LIN {X 0,Y 472.91,Z 456.577,A -85,B 0,C 180,E1 22479.324,E2 22479.324} C_VEL
LIN {X 0,Y 472.927,Z 456.575,A -85,B 0,C 180,E1 22475.519,E2 22475.519} C_VEL
LIN {X 0,Y 472.958,Z 456.569,A -85,B 0,C 180,E1 22471.872,E2 22471.872} C_VEL
LIN {X 0,Y 472.951,Z 456.569,A -85,B 0,C 180,E1 22468.195,E2 22468.195} C_VEL
LIN {X 0,Y 472.938,Z 456.573,A -85,B 0,C 180,E1 22464.6,E2 22464.6} C_VEL
LIN {X 0,Y 472.903,Z 456.579,A -85,B 0,C 180,E1 22460.89,E2 22460.89} C_VEL
LIN {X 0,Y 472.947,Z 456.574,A -85,B 0,C 180,E1 22457.263,E2 22457.263} C_VEL
LIN {X 0,Y 472.93,Z 456.574,A -85,B 0,C 180,E1 22453.693,E2 22453.693} C_VEL
LIN {X 0,Y 472.947,Z 456.701,A -85,B 0,C 180,E1 22450.415,E2 22450.415} C_VEL
LIN {X 0,Y 481.637,Z 478.377,A -85,B 0,C 180,E1 22447.531,E2 22447.531} C_VEL
LIN {X 0,Y 487.148,Z 493.23,A -85,B 0,C 180,E1 22445.727,E2 22445.727} C_VEL
LIN {X 0,Y 487.147,Z 498.207,A -85,B 0,C 180,E1 22445.36,E2 22445.36} C_VEL
LIN {X 0,Y 491.021,Z 519.873,A -85,B 0,C 180,E1 22444.656,E2 22444.656} C_VEL
LIN {X 0,Y 490.363,Z 557.478,A -85,B 0,C 180,E1 22444.053,E2 22444.053} C_VEL
LIN {X 0,Y 489.42,Z 565.168,A -85,B 0,C 180,E1 22443.994,E2 22443.994} C_VEL
LIN {X 0,Y 483.858,Z 585.669,A -85,B 0,C 180,E1 22444.081,E2 22444.081} C_VEL
LIN {X 0,Y 483.117,Z 592.27,A -85,B 0,C 180,E1 22444.025,E2 22444.025} C_VEL
LIN {X 0,Y 480.112,Z 758.652,A -85,B 0,C 180,E1 22441.318,E2 22441.318} C_VEL
LIN {X 0,Y 479.264,Z 779.44,A -85,B 0,C 180,E1 22440.773,E2 22440.773} C_VEL
LIN {X 0,Y 478.093,Z 800.27,A -85,B 0,C 180,E1 22439.988,E2 22439.988} C_VEL
LIN {X 0,Y 476.733,Z 819.282,A -85,B 0,C 180,E1 22439.046,E2 22439.046} C_VEL
LIN {X 0,Y 475.203,Z 837.681,A -85,B 0,C 180,E1 22437.907,E2 22437.907} C_VEL
LIN {X 0,Y 473.52,Z 855.537,A -85,B 0,C 180,E1 22436.551,E2 22436.551} C_VEL
LIN {X 0,Y 471.822,Z 872.211,A -85,B 0,C 180,E1 22435.024,E2 22435.024} C_VEL
LIN {X 0,Y 470.132,Z 888.047,A -85,B 0,C 180,E1 22433.301,E2 22433.301} C_VEL
LIN {X 0,Y 468.579,Z 902.793,A -85,B 0,C 180,E1 22431.4,E2 22431.4} C_VEL
LIN {X 0,Y 467.185,Z 916.53,A -85,B 0,C 180,E1 22429.296,E2 22429.296} C_VEL
LIN {X 0,Y 466.056,Z 928.61,A -85,B 0,C 180,E1 22427.092,E2 22427.092} C_VEL
LIN {X 0,Y 465.206,Z 939.007,A -85,B 0,C 180,E1 22424.818,E2 22424.818} C_VEL
LIN {X 0,Y 464.592,Z 947.948,A -85,B 0,C 180,E1 22422.427,E2 22422.427} C_VEL
LIN {X 0,Y 464.221,Z 955.037,A -85,B 0,C 180,E1 22420.047,E2 22420.047} C_VEL
LIN {X 0,Y 464.015,Z 960.75,A -85,B 0,C 180,E1 22417.552,E2 22417.552} C_VEL
LIN {X 0,Y 463.931,Z 964.938,A -85,B 0,C 180,E1 22414.945,E2 22414.945} C_VEL
LIN {X 0,Y 463.912,Z 967.307,A -85,B 0,C 180,E1 22412.47,E2 22412.47} C_VEL
LIN {X 0,Y 463.915,Z 968.138,A -85,B 0,C 180,E1 22409.999,E2 22409.999} C_VEL
LIN {X 0,Y 463.908,Z 967.355,A -85,B 0,C 180,E1 22407.529,E2 22407.529} C_VEL
LIN {X 0,Y 463.932,Z 965.05,A -85,B 0,C 180,E1 22405.054,E2 22405.054} C_VEL
LIN {X 0,Y 464.002,Z 961.169,A -85,B 0,C 180,E1 22402.571,E2 22402.571} C_VEL
LIN {X 0,Y 464.188,Z 955.956,A -85,B 0,C 180,E1 22400.202,E2 22400.202} C_VEL
LIN {X 0,Y 464.549,Z 948.649,A -85,B 0,C 180,E1 22397.696,E2 22397.696} C_VEL
LIN {X 0,Y 465.133,Z 939.852,A -85,B 0,C 180,E1 22395.305,E2 22395.305} C_VEL
LIN {X 0,Y 465.959,Z 929.65,A -85,B 0,C 180,E1 22393.032,E2 22393.032} C_VEL
LIN {X 0,Y 467.101,Z 917.348,A -85,B 0,C 180,E1 22390.752,E2 22390.752} C_VEL
LIN {X 0,Y 468.516,Z 903.403,A -85,B 0,C 180,E1 22388.596,E2 22388.596} C_VEL
LIN {X 0,Y 470.064,Z 888.771,A -85,B 0,C 180,E1 22386.694,E2 22386.694} C_VEL
LIN {X 0,Y 471.702,Z 873.45,A -85,B 0,C 180,E1 22385.007,E2 22385.007} C_VEL
LIN {X 0,Y 473.47,Z 856.09,A -85,B 0,C 180,E1 22383.403,E2 22383.403} C_VEL
LIN {X 0,Y 475.187,Z 837.858,A -85,B 0,C 180,E1 22382.015,E2 22382.015} C_VEL
LIN {X 0,Y 476.704,Z 819.608,A -85,B 0,C 180,E1 22380.881,E2 22380.881} C_VEL
LIN {X 0,Y 478.069,Z 800.671,A -85,B 0,C 180,E1 22379.94,E2 22379.94} C_VEL
LIN {X 0,Y 479.224,Z 780.234,A -85,B 0,C 180,E1 22379.162,E2 22379.162} C_VEL
LIN {X 0,Y 480.082,Z 759.903,A -85,B 0,C 180,E1 22378.618,E2 22378.618} C_VEL
LIN {X 0,Y 481.257,Z 696.258,A -85,B 0,C 180,E1 22377.561,E2 22377.561} C_VEL
LIN {X 0,Y 484.181,Z 528.146,A -85,B 0,C 180,E1 22374.833,E2 22374.833} C_VEL
LIN {X 0,Y 476.532,Z 500.148,A -85,B 0,C 180,E1 22373.647,E2 22373.647} C_VEL
LIN {X 0,Y 476.698,Z 493.601,A -85,B 0,C 180,E1 22372.837,E2 22372.837} C_VEL
LIN {X 0,Y 471.955,Z 477.879,A -85,B 0,C 180,E1 22370.222,E2 22370.222} C_VEL
LIN {X 0,Y 466.792,Z 462.968,A -85,B 0,C 180,E1 22367.566,E2 22367.566} C_VEL
LIN {X 0,Y 465.01,Z 457.558,A -85,B 0,C 180,E1 22366.565,E2 22366.565} C_VEL
LIN {X 0,Y 465.012,Z 457.562,A -85,B 0,C 180,E1 22362.843,E2 22362.843} C_VEL
LIN {X 0,Y 465.017,Z 457.564,A -85,B 0,C 180,E1 22359.209,E2 22359.209} C_VEL
LIN {X 0,Y 465.008,Z 457.58,A -85,B 0,C 180,E1 22355.73,E2 22355.73} C_VEL
LIN {X 0,Y 473.084,Z 479.715,A -85,B 0,C 180,E1 22352.397,E2 22352.397} C_VEL
LIN {X 0,Y 478.097,Z 494.806,A -85,B 0,C 180,E1 22350.262,E2 22350.262} C_VEL
LIN {X 0,Y 476.18,Z 526.834,A -85,B 0,C 180,E1 22346.904,E2 22346.904} C_VEL
LIN {X 0,Y 474.134,Z 562.551,A -85,B 0,C 180,E1 22343.226,E2 22343.226} C_VEL
LIN {X 0,Y 472.412,Z 597.934,A -85,B 0,C 180,E1 22339.635,E2 22339.635} C_VEL
LIN {X 0,Y 471.717,Z 615.117,A -85,B 0,C 180,E1 22337.947,E2 22337.947} C_VEL
LIN {X 0,Y 472.395,Z 621.151,A -85,B 0,C 180,E1 22337.789,E2 22337.789} C_VEL
LIN {X 0,Y 469.651,Z 757.732,A -85,B 0,C 180,E1 22335.181,E2 22335.181} C_VEL
LIN {X 0,Y 469.368,Z 774.573,A -85,B 0,C 180,E1 22334.622,E2 22334.622} C_VEL
LIN {X 0,Y 468.917,Z 789.931,A -85,B 0,C 180,E1 22333.88,E2 22333.88} C_VEL
LIN {X 0,Y 468.342,Z 805.227,A -85,B 0,C 180,E1 22332.891,E2 22332.891} C_VEL
LIN {X 0,Y 467.722,Z 818.619,A -85,B 0,C 180,E1 22331.78,E2 22331.78} C_VEL
LIN {X 0,Y 467.018,Z 832.225,A -85,B 0,C 180,E1 22330.361,E2 22330.361} C_VEL
LIN {X 0,Y 466.406,Z 843.527,A -85,B 0,C 180,E1 22328.879,E2 22328.879} C_VEL
LIN {X 0,Y 465.85,Z 854.094,A -85,B 0,C 180,E1 22327.151,E2 22327.151} C_VEL
LIN {X 0,Y 465.438,Z 862.373,A -85,B 0,C 180,E1 22325.424,E2 22325.424} C_VEL
LIN {X 0,Y 465.125,Z 869.663,A -85,B 0,C 180,E1 22323.451,E2 22323.451} C_VEL
LIN {X 0,Y 464.929,Z 874.839,A -85,B 0,C 180,E1 22321.479,E2 22321.479} C_VEL
LIN {X 0,Y 464.858,Z 878.245,A -85,B 0,C 180,E1 22319.507,E2 22319.507} C_VEL
LIN {X 0,Y 464.842,Z 879.886,A -85,B 0,C 180,E1 22317.535,E2 22317.535} C_VEL
LIN {X 0,Y 464.923,Z 879.826,A -85,B 0,C 180,E1 22315.436,E2 22315.436} C_VEL
LIN {X 0,Y 465.055,Z 877.967,A -85,B 0,C 180,E1 22313.457,E2 22313.457} C_VEL
LIN {X 0,Y 465.317,Z 874.396,A -85,B 0,C 180,E1 22311.474,E2 22311.474} C_VEL
LIN {X 0,Y 465.678,Z 869.023,A -85,B 0,C 180,E1 22309.541,E2 22309.541} C_VEL
LIN {X 0,Y 466.158,Z 862.251,A -85,B 0,C 180,E1 22307.74,E2 22307.74} C_VEL
LIN {X 0,Y 466.757,Z 853.636,A -85,B 0,C 180,E1 22305.992,E2 22305.992} C_VEL
LIN {X 0,Y 467.47,Z 843.493,A -85,B 0,C 180,E1 22304.366,E2 22304.366} C_VEL
LIN {X 0,Y 468.204,Z 832.087,A -85,B 0,C 180,E1 22302.925,E2 22302.925} C_VEL
LIN {X 0,Y 468.927,Z 819.784,A -85,B 0,C 180,E1 22301.669,E2 22301.669} C_VEL
LIN {X 0,Y 469.544,Z 806.42,A -85,B 0,C 180,E1 22300.598,E2 22300.598} C_VEL
LIN {X 0,Y 470.043,Z 792.265,A -85,B 0,C 180,E1 22299.713,E2 22299.713} C_VEL
LIN {X 0,Y 470.359,Z 776.806,A -85,B 0,C 180,E1 22299.011,E2 22299.011} C_VEL
LIN {X 0,Y 470.464,Z 760.839,A -85,B 0,C 180,E1 22298.522,E2 22298.522} C_VEL
LIN {X 0,Y 472.137,Z 707.062,A -85,B 0,C 180,E1 22297.264,E2 22297.264} C_VEL
LIN {X 0,Y 475.823,Z 635.91,A -85,B 0,C 180,E1 22295.48,E2 22295.48} C_VEL
LIN {X 0,Y 479.671,Z 625.998,A -85,B 0,C 180,E1 22294.637,E2 22294.637} C_VEL
LIN {X 0,Y 484.504,Z 596.236,A -85,B 0,C 180,E1 22290.99,E2 22290.99} C_VEL
LIN {X 0,Y 490.347,Z 571.27,A -85,B 0,C 180,E1 22287.708,E2 22287.708} C_VEL
LIN {X 0,Y 496.915,Z 551.415,A -85,B 0,C 180,E1 22284.868,E2 22284.868} C_VEL
LIN {X 0,Y 504.072,Z 536.502,A -85,B 0,C 180,E1 22282.508,E2 22282.508} C_VEL
LIN {X 0,Y 506.427,Z 532.598,A -85,B 0,C 180,E1 22281.76,E2 22281.76} C_VEL
LIN {X 0,Y 506.709,Z 532.003,A -85,B 0,C 180,E1 22281.259,E2 22281.259} C_VEL
LIN {X 0,Y 498.452,Z 544.531,A -85,B 0,C 180,E1 22279.664,E2 22279.664} C_VEL
LIN {X 0,Y 491.821,Z 558.642,A -85,B 0,C 180,E1 22278.022,E2 22278.022} C_VEL
LIN {X 0,Y 487.188,Z 573.707,A -85,B 0,C 180,E1 22276.34,E2 22276.34} C_VEL
LIN {X 0,Y 484.882,Z 588.959,A -85,B 0,C 180,E1 22274.65,E2 22274.65} C_VEL
LIN {X 0,Y 484.928,Z 602.549,A -85,B 0,C 180,E1 22273.122,E2 22273.122} C_VEL
LIN {X 0,Y 487.165,Z 615.999,A -85,B 0,C 180,E1 22271.574,E2 22271.574} C_VEL
LIN {X 0,Y 491.226,Z 627.81,A -85,B 0,C 180,E1 22270.184,E2 22270.184} C_VEL
LIN {X 0,Y 497.098,Z 638.674,A -85,B 0,C 180,E1 22268.871,E2 22268.871} C_VEL
LIN {X 0,Y 504.869,Z 648.854,A -85,B 0,C 180,E1 22267.611,E2 22267.611} C_VEL
LIN {X 0,Y 514.493,Z 658.204,A -85,B 0,C 180,E1 22266.432,E2 22266.432} C_VEL
LIN {X 0,Y 526.445,Z 666.953,A -85,B 0,C 180,E1 22265.302,E2 22265.302} C_VEL
LIN {X 0,Y 516.888,Z 683.64,A -85,B 0,C 180,E1 22264.661,E2 22264.661} C_VEL
LIN {X 0,Y 504.016,Z 702.431,A -85,B 0,C 180,E1 22264.017,E2 22264.017} C_VEL
LIN {X 0,Y 495.13,Z 717.971,A -85,B 0,C 180,E1 22263.387,E2 22263.387} C_VEL
LIN {X 0,Y 488.588,Z 732.528,A -85,B 0,C 180,E1 22262.702,E2 22262.702} C_VEL
LIN {X 0,Y 482.078,Z 749.198,A -85,B 0,C 180,E1 22261.887,E2 22261.887} C_VEL
LIN {X 0,Y 479.563,Z 772.367,A -85,B 0,C 180,E1 22261.674,E2 22261.674} C_VEL
LIN {X 0,Y 478.792,Z 805.933,A -85,B 0,C 180,E1 22261.099,E2 22261.099} C_VEL
LIN {X 0,Y 477.845,Z 826.58,A -85,B 0,C 180,E1 22260.534,E2 22260.534} C_VEL
LIN {X 0,Y 476.592,Z 846.828,A -85,B 0,C 180,E1 22259.747,E2 22259.747} C_VEL
LIN {X 0,Y 475.191,Z 866.116,A -85,B 0,C 180,E1 22258.765,E2 22258.765} C_VEL
LIN {X 0,Y 473.67,Z 884.493,A -85,B 0,C 180,E1 22257.603,E2 22257.603} C_VEL
LIN {X 0,Y 472.077,Z 902.359,A -85,B 0,C 180,E1 22256.233,E2 22256.233} C_VEL
LIN {X 0,Y 470.518,Z 919.286,A -85,B 0,C 180,E1 22254.682,E2 22254.682} C_VEL
LIN {X 0,Y 469.001,Z 935.399,A -85,B 0,C 180,E1 22252.931,E2 22252.931} C_VEL
LIN {X 0,Y 467.587,Z 950.936,A -85,B 0,C 180,E1 22250.923,E2 22250.923} C_VEL
LIN {X 0,Y 466.486,Z 964.207,A -85,B 0,C 180,E1 22248.885,E2 22248.885} C_VEL
LIN {X 0,Y 465.557,Z 976.373,A -85,B 0,C 180,E1 22246.694,E2 22246.694} C_VEL
LIN {X 0,Y 464.832,Z 988.822,A -85,B 0,C 180,E1 22244.068,E2 22244.068} C_VEL
LIN {X 0,Y 464.446,Z 996.901,A -85,B 0,C 180,E1 22242.054,E2 22242.054} C_VEL
LIN {X 0,Y 464.164,Z 1004.554,A -85,B 0,C 180,E1 22239.673,E2 22239.673} C_VEL
LIN {X 0,Y 464.004,Z 1009.721,A -85,B 0,C 180,E1 22237.595,E2 22237.595} C_VEL
LIN {X 0,Y 463.928,Z 1013.749,A -85,B 0,C 180,E1 22235.442,E2 22235.442} C_VEL
LIN {X 0,Y 463.909,Z 1016.649,A -85,B 0,C 180,E1 22232.966,E2 22232.966} C_VEL
LIN {X 0,Y 463.909,Z 1017.726,A -85,B 0,C 180,E1 22230.865,E2 22230.865} C_VEL
LIN {X 0,Y 463.902,Z 1017.607,A -85,B 0,C 180,E1 22228.642,E2 22228.642} C_VEL
LIN {X 0,Y 463.919,Z 1015.695,A -85,B 0,C 180,E1 22226.046,E2 22226.046} C_VEL
LIN {X 0,Y 463.956,Z 1012.73,A -85,B 0,C 180,E1 22223.939,E2 22223.939} C_VEL
LIN {X 0,Y 464.064,Z 1007.975,A -85,B 0,C 180,E1 22221.576,E2 22221.576} C_VEL
LIN {X 0,Y 464.27,Z 1001.352,A -85,B 0,C 180,E1 22219.202,E2 22219.202} C_VEL
LIN {X 0,Y 464.574,Z 994.236,A -85,B 0,C 180,E1 22217.148,E2 22217.148} C_VEL
LIN {X 0,Y 465.136,Z 983.695,A -85,B 0,C 180,E1 22214.669,E2 22214.669} C_VEL
LIN {X 0,Y 465.804,Z 973.255,A -85,B 0,C 180,E1 22212.641,E2 22212.641} C_VEL
LIN {X 0,Y 466.988,Z 957.492,A -85,B 0,C 180,E1 22210.04,E2 22210.04} C_VEL
LIN {X 0,Y 468.228,Z 943.394,A -85,B 0,C 180,E1 22208.057,E2 22208.057} C_VEL
LIN {X 0,Y 469.719,Z 927.266,A -85,B 0,C 180,E1 22206.145,E2 22206.145} C_VEL
LIN {X 0,Y 471.349,Z 909.972,A -85,B 0,C 180,E1 22204.427,E2 22204.427} C_VEL
LIN {X 0,Y 472.911,Z 892.363,A -85,B 0,C 180,E1 22202.964,E2 22202.964} C_VEL
LIN {X 0,Y 474.503,Z 873.954,A -85,B 0,C 180,E1 22201.699,E2 22201.699} C_VEL
LIN {X 0,Y 476.021,Z 854.172,A -85,B 0,C 180,E1 22200.599,E2 22200.599} C_VEL
LIN {X 0,Y 477.32,Z 834.383,A -85,B 0,C 180,E1 22199.741,E2 22199.741} C_VEL
LIN {X 0,Y 478.39,Z 814.17,A -85,B 0,C 180,E1 22199.095,E2 22199.095} C_VEL
LIN {X 0,Y 479.108,Z 792.718,A -85,B 0,C 180,E1 22198.642,E2 22198.642} C_VEL
LIN {X 0,Y 479.824,Z 766.954,A -85,B 0,C 180,E1 22198.252,E2 22198.252} C_VEL
LIN {X 0,Y 480.143,Z 763.831,A -85,B 0,C 180,E1 22198.208,E2 22198.208} C_VEL
LIN {X 0,Y 485.952,Z 747.066,A -85,B 0,C 180,E1 22197.302,E2 22197.302} C_VEL
LIN {X 0,Y 495.745,Z 723.845,A -85,B 0,C 180,E1 22196.197,E2 22196.197} C_VEL
LIN {X 0,Y 504.216,Z 708.095,A -85,B 0,C 180,E1 22195.588,E2 22195.588} C_VEL
LIN {X 0,Y 516.218,Z 689.456,A -85,B 0,C 180,E1 22195.015,E2 22195.015} C_VEL
LIN {X 0,Y 520.11,Z 683.607,A -85,B 0,C 180,E1 22194.848,E2 22194.848} C_VEL
LIN {X 0,Y 528.054,Z 668.908,A -85,B 0,C 180,E1 22194.321,E2 22194.321} C_VEL
LIN {X 0,Y 516.85,Z 661.041,A -85,B 0,C 180,E1 22193.013,E2 22193.013} C_VEL
LIN {X 0,Y 507.468,Z 651.762,A -85,B 0,C 180,E1 22191.644,E2 22191.644} C_VEL
LIN {X 0,Y 500.207,Z 641.723,A -85,B 0,C 180,E1 22190.315,E2 22190.315} C_VEL
LIN {X 0,Y 494.469,Z 630.437,A -85,B 0,C 180,E1 22188.959,E2 22188.959} C_VEL
LIN {X 0,Y 490.186,Z 617.3,A -85,B 0,C 180,E1 22187.534,E2 22187.534} C_VEL
LIN {X 0,Y 487.49,Z 602.313,A -85,B 0,C 180,E1 22186.047,E2 22186.047} C_VEL
LIN {X 0,Y 486.582,Z 585.023,A -85,B 0,C 180,E1 22184.484,E2 22184.484} C_VEL
LIN {X 0,Y 487.699,Z 561.885,A -85,B 0,C 180,E1 22182.574,E2 22182.574} C_VEL
LIN {X 0,Y 490.859,Z 525.783,A -85,B 0,C 180,E1 22179.65,E2 22179.65} C_VEL
LIN {X 0,Y 492.028,Z 513.047,A -85,B 0,C 180,E1 22178.598,E2 22178.598} C_VEL
LIN {X 0,Y 482.947,Z 494.174,A -85,B 0,C 180,E1 22175.72,E2 22175.72} C_VEL
LIN {X 0,Y 473.608,Z 475.089,A -85,B 0,C 180,E1 22172.571,E2 22172.571} C_VEL
LIN {X 0,Y 468.839,Z 465.842,A -85,B 0,C 180,E1 22170.928,E2 22170.928} C_VEL
LIN {X 0,Y 466.513,Z 461.325,A -85,B 0,C 180,E1 22170.101,E2 22170.101} C_VEL
LIN {X 0,Y 465.011,Z 457.678,A -85,B 0,C 180,E1 22169.478,E2 22169.478} C_VEL
LIN {X 0,Y 465.009,Z 457.562,A -85,B 0,C 180,E1 22165.743,E2 22165.743} C_VEL
LIN {X 0,Y 464.994,Z 457.565,A -85,B 0,C 180,E1 22162.104,E2 22162.104} C_VEL
LIN {X 0,Y 464.979,Z 457.567,A -85,B 0,C 180,E1 22158.427,E2 22158.427} C_VEL
LIN {X 0,Y 465.016,Z 457.563,A -85,B 0,C 180,E1 22154.825,E2 22154.825} C_VEL
LIN {X 0,Y 464.988,Z 457.566,A -85,B 0,C 180,E1 22151.158,E2 22151.158} C_VEL
LIN {X 0,Y 465.011,Z 457.561,A -85,B 0,C 180,E1 22147.536,E2 22147.536} C_VEL
LIN {X 0,Y 464.963,Z 457.568,A -85,B 0,C 180,E1 22143.946,E2 22143.946} C_VEL
LIN {X 0,Y 464.993,Z 457.562,A -85,B 0,C 180,E1 22140.246,E2 22140.246} C_VEL
LIN {X 0,Y 465.013,Z 457.564,A -85,B 0,C 180,E1 22136.672,E2 22136.672} C_VEL
LIN {X 0,Y 465.017,Z 457.548,A -85,B 0,C 180,E1 22132.836,E2 22132.836} C_VEL
LIN {X 0,Y 464.994,Z 457.563,A -85,B 0,C 180,E1 22129.218,E2 22129.218} C_VEL
LIN {X 0,Y 464.967,Z 457.562,A -85,B 0,C 180,E1 22125.428,E2 22125.428} C_VEL
LIN {X 0,Y 465.008,Z 457.55,A -85,B 0,C 180,E1 22121.833,E2 22121.833} C_VEL
LIN {X 0,Y 465.003,Z 457.555,A -85,B 0,C 180,E1 22118.162,E2 22118.162} C_VEL
LIN {X 0,Y 465.013,Z 457.561,A -85,B 0,C 180,E1 22114.53,E2 22114.53} C_VEL
LIN {X 0,Y 464.97,Z 457.568,A -85,B 0,C 180,E1 22110.923,E2 22110.923} C_VEL
LIN {X 0,Y 464.988,Z 457.566,A -85,B 0,C 180,E1 22107.189,E2 22107.189} C_VEL
LIN {X 0,Y 465.016,Z 457.565,A -85,B 0,C 180,E1 22103.528,E2 22103.528} C_VEL
LIN {X 0,Y 465.022,Z 457.556,A -85,B 0,C 180,E1 22099.755,E2 22099.755} C_VEL
LIN {X 0,Y 464.998,Z 457.561,A -85,B 0,C 180,E1 22096.081,E2 22096.081} C_VEL
LIN {X 0,Y 464.967,Z 457.569,A -85,B 0,C 180,E1 22092.291,E2 22092.291} C_VEL
LIN {X 0,Y 465.006,Z 457.62,A -85,B 0,C 180,E1 22091.144,E2 22091.144} C_VEL
LIN {X 0,Y 466.275,Z 461.028,A -85,B 0,C 180,E1 22090.683,E2 22090.683} C_VEL
LIN {X 0,Y 473.647,Z 478.764,A -85,B 0,C 180,E1 22088.253,E2 22088.253} C_VEL
LIN {X 0,Y 480.276,Z 496.419,A -85,B 0,C 180,E1 22086.077,E2 22086.077} C_VEL
LIN {X 0,Y 480.45,Z 498.811,A -85,B 0,C 180,E1 22085.923,E2 22085.923} C_VEL
LIN {X 0,Y 484.443,Z 521.253,A -85,B 0,C 180,E1 22085.177,E2 22085.177} C_VEL
LIN {X 0,Y 483.117,Z 592.27,A -85,B 0,C 180,E1 22084.025,E2 22084.025} C_VEL
LIN {X 0,Y 482.157,Z 599.961,A -85,B 0,C 180,E1 22083.966,E2 22083.966} C_VEL
LIN {X 0,Y 476.58,Z 620.456,A -85,B 0,C 180,E1 22084.055,E2 22084.055} C_VEL
LIN {X 0,Y 475.826,Z 627.058,A -85,B 0,C 180,E1 22083.999,E2 22083.999} C_VEL
LIN {X 0,Y 473.287,Z 759.334,A -85,B 0,C 180,E1 22081.813,E2 22081.813} C_VEL
LIN {X 0,Y 472.398,Z 779.954,A -85,B 0,C 180,E1 22081.264,E2 22081.264} C_VEL
LIN {X 0,Y 471.167,Z 800.633,A -85,B 0,C 180,E1 22080.475,E2 22080.475} C_VEL
LIN {X 0,Y 469.702,Z 819.966,A -85,B 0,C 180,E1 22079.504,E2 22079.504} C_VEL
LIN {X 0,Y 468.075,Z 838.339,A -85,B 0,C 180,E1 22078.348,E2 22078.348} C_VEL
LIN {X 0,Y 466.286,Z 856.248,A -85,B 0,C 180,E1 22076.968,E2 22076.968} C_VEL
LIN {X 0,Y 464.421,Z 873.405,A -85,B 0,C 180,E1 22075.367,E2 22075.367} C_VEL
LIN {X 0,Y 462.695,Z 888.451,A -85,B 0,C 180,E1 22073.699,E2 22073.699} C_VEL
LIN {X 0,Y 461.032,Z 903.202,A -85,B 0,C 180,E1 22071.768,E2 22071.768} C_VEL
LIN {X 0,Y 459.575,Z 916.502,A -85,B 0,C 180,E1 22069.707,E2 22069.707} C_VEL
LIN {X 0,Y 458.366,Z 928.408,A -85,B 0,C 180,E1 22067.519,E2 22067.519} C_VEL
LIN {X 0,Y 457.418,Z 938.91,A -85,B 0,C 180,E1 22065.206,E2 22065.206} C_VEL
LIN {X 0,Y 456.728,Z 947.92,A -85,B 0,C 180,E1 22062.773,E2 22062.773} C_VEL
LIN {X 0,Y 456.29,Z 955.25,A -85,B 0,C 180,E1 22060.299,E2 22060.299} C_VEL
LIN {X 0,Y 456.064,Z 960.918,A -85,B 0,C 180,E1 22057.812,E2 22057.812} C_VEL
LIN {X 0,Y 455.949,Z 965.044,A -85,B 0,C 180,E1 22055.284,E2 22055.284} C_VEL
LIN {X 0,Y 455.926,Z 967.588,A -85,B 0,C 180,E1 22052.765,E2 22052.765} C_VEL
LIN {X 0,Y 455.925,Z 968.528,A -85,B 0,C 180,E1 22050.125,E2 22050.125} C_VEL
LIN {X 0,Y 455.92,Z 967.832,A -85,B 0,C 180,E1 22047.611,E2 22047.611} C_VEL
LIN {X 0,Y 455.948,Z 965.462,A -85,B 0,C 180,E1 22044.967,E2 22044.967} C_VEL
LIN {X 0,Y 456.035,Z 961.58,A -85,B 0,C 180,E1 22042.44,E2 22042.44} C_VEL
LIN {X 0,Y 456.247,Z 956.368,A -85,B 0,C 180,E1 22040.03,E2 22040.03} C_VEL
LIN {X 0,Y 456.649,Z 949.061,A -85,B 0,C 180,E1 22037.48,E2 22037.48} C_VEL
LIN {X 0,Y 457.295,Z 940.262,A -85,B 0,C 180,E1 22035.048,E2 22035.048} C_VEL
LIN {X 0,Y 458.195,Z 930.057,A -85,B 0,C 180,E1 22032.735,E2 22032.735} C_VEL
LIN {X 0,Y 459.435,Z 917.751,A -85,B 0,C 180,E1 22030.418,E2 22030.418} C_VEL
LIN {X 0,Y 460.965,Z 903.801,A -85,B 0,C 180,E1 22028.228,E2 22028.228} C_VEL
LIN {X 0,Y 462.668,Z 888.727,A -85,B 0,C 180,E1 22026.244,E2 22026.244} C_VEL
LIN {X 0,Y 464.468,Z 872.95,A -85,B 0,C 180,E1 22024.497,E2 22024.497} C_VEL
LIN {X 0,Y 466.265,Z 856.46,A -85,B 0,C 180,E1 22022.959,E2 22022.959} C_VEL
LIN {X 0,Y 468.09,Z 838.221,A -85,B 0,C 180,E1 22021.553,E2 22021.553} C_VEL
LIN {X 0,Y 469.703,Z 819.96,A -85,B 0,C 180,E1 22020.405,E2 22020.405} C_VEL
LIN {X 0,Y 471.159,Z 800.795,A -85,B 0,C 180,E1 22019.442,E2 22019.442} C_VEL
LIN {X 0,Y 472.394,Z 780.039,A -85,B 0,C 180,E1 22018.648,E2 22018.648} C_VEL
LIN {X 0,Y 473.289,Z 759.337,A -85,B 0,C 180,E1 22018.097,E2 22018.097} C_VEL
LIN {X 0,Y 476.178,Z 607.269,A -85,B 0,C 180,E1 22015.583,E2 22015.583} C_VEL
LIN {X 0,Y 477.536,Z 529.583,A -85,B 0,C 180,E1 22014.292,E2 22014.292} C_VEL
LIN {X 0,Y 469.619,Z 500.423,A -85,B 0,C 180,E1 22013.017,E2 22013.017} C_VEL
LIN {X 0,Y 469.622,Z 496.818,A -85,B 0,C 180,E1 22012.575,E2 22012.575} C_VEL
LIN {X 0,Y 464.912,Z 481.204,A -85,B 0,C 180,E1 22009.963,E2 22009.963} C_VEL
LIN {X 0,Y 459.304,Z 464.811,A -85,B 0,C 180,E1 22007.007,E2 22007.007} C_VEL
LIN {X 0,Y 457.05,Z 458.55,A -85,B 0,C 180,E1 22005.797,E2 22005.797} C_VEL
LIN {X 0,Y 457.06,Z 458.547,A -85,B 0,C 180,E1 22002.021,E2 22002.021} C_VEL
LIN {X 0,Y 457.074,Z 458.552,A -85,B 0,C 180,E1 21998.408,E2 21998.408} C_VEL
LIN {X 0,Y 457.096,Z 458.744,A -85,B 0,C 180,E1 21996.392,E2 21996.392} C_VEL
LIN {X 0,Y 465.159,Z 480.489,A -85,B 0,C 180,E1 21993.037,E2 21993.037} C_VEL
LIN {X 0,Y 470.961,Z 497.618,A -85,B 0,C 180,E1 21990.562,E2 21990.562} C_VEL
LIN {X 0,Y 468.998,Z 528.902,A -85,B 0,C 180,E1 21987.25,E2 21987.25} C_VEL
LIN {X 0,Y 466.848,Z 564.434,A -85,B 0,C 180,E1 21983.556,E2 21983.556} C_VEL
LIN {X 0,Y 465.013,Z 599.849,A -85,B 0,C 180,E1 21979.926,E2 21979.926} C_VEL
LIN {X 0,Y 464.303,Z 616.005,A -85,B 0,C 180,E1 21978.32,E2 21978.32} C_VEL
LIN {X 0,Y 465.008,Z 622.209,A -85,B 0,C 180,E1 21978.154,E2 21978.154} C_VEL
LIN {X 0,Y 462.034,Z 758.851,A -85,B 0,C 180,E1 21975.461,E2 21975.461} C_VEL
LIN {X 0,Y 461.725,Z 775.984,A -85,B 0,C 180,E1 21974.877,E2 21974.877} C_VEL
LIN {X 0,Y 461.246,Z 791.353,A -85,B 0,C 180,E1 21974.115,E2 21974.115} C_VEL
LIN {X 0,Y 460.641,Z 806.561,A -85,B 0,C 180,E1 21973.11,E2 21973.11} C_VEL
LIN {X 0,Y 459.952,Z 820.55,A -85,B 0,C 180,E1 21971.918,E2 21971.918} C_VEL
LIN {X 0,Y 459.245,Z 833.485,A -85,B 0,C 180,E1 21970.538,E2 21970.538} C_VEL
LIN {X 0,Y 458.587,Z 844.985,A -85,B 0,C 180,E1 21969,E2 21969} C_VEL
LIN {X 0,Y 458.01,Z 855.345,A -85,B 0,C 180,E1 21967.274,E2 21967.274} C_VEL
LIN {X 0,Y 457.572,Z 863.623,A -85,B 0,C 180,E1 21965.517,E2 21965.517} C_VEL
LIN {X 0,Y 457.239,Z 870.93,A -85,B 0,C 180,E1 21963.511,E2 21963.511} C_VEL
LIN {X 0,Y 457.032,Z 876.115,A -85,B 0,C 180,E1 21961.505,E2 21961.505} C_VEL
LIN {X 0,Y 456.958,Z 879.536,A -85,B 0,C 180,E1 21959.499,E2 21959.499} C_VEL
LIN {X 0,Y 456.946,Z 881.179,A -85,B 0,C 180,E1 21957.492,E2 21957.492} C_VEL
LIN {X 0,Y 457.038,Z 881.126,A -85,B 0,C 180,E1 21955.357,E2 21955.357} C_VEL
LIN {X 0,Y 457.194,Z 879.271,A -85,B 0,C 180,E1 21953.344,E2 21953.344} C_VEL
LIN {X 0,Y 457.49,Z 875.714,A -85,B 0,C 180,E1 21951.327,E2 21951.327} C_VEL
LIN {X 0,Y 457.879,Z 870.565,A -85,B 0,C 180,E1 21949.431,E2 21949.431} C_VEL
LIN {X 0,Y 458.429,Z 863.572,A -85,B 0,C 180,E1 21947.53,E2 21947.53} C_VEL
LIN {X 0,Y 459.088,Z 854.863,A -85,B 0,C 180,E1 21945.74,E2 21945.74} C_VEL
LIN {X 0,Y 459.864,Z 844.801,A -85,B 0,C 180,E1 21944.1,E2 21944.1} C_VEL
LIN {X 0,Y 460.709,Z 832.889,A -85,B 0,C 180,E1 21942.573,E2 21942.573} C_VEL
LIN {X 0,Y 461.444,Z 821.109,A -85,B 0,C 180,E1 21941.361,E2 21941.361} C_VEL
LIN {X 0,Y 462.144,Z 806.943,A -85,B 0,C 180,E1 21940.216,E2 21940.216} C_VEL
LIN {X 0,Y 462.661,Z 793.229,A -85,B 0,C 180,E1 21939.353,E2 21939.353} C_VEL
LIN {X 0,Y 463.025,Z 776.838,A -85,B 0,C 180,E1 21938.605,E2 21938.605} C_VEL
LIN {X 0,Y 463.119,Z 759.97,A -85,B 0,C 180,E1 21938.105,E2 21938.105} C_VEL
LIN {X 0,Y 465.355,Z 702.161,A -85,B 0,C 180,E1 21936.667,E2 21936.667} C_VEL
LIN {X 0,Y 469.061,Z 638.911,A -85,B 0,C 180,E1 21935.002,E2 21935.002} C_VEL
LIN {X 0,Y 473.322,Z 628.666,A -85,B 0,C 180,E1 21934.146,E2 21934.146} C_VEL
LIN {X 0,Y 478.491,Z 599.761,A -85,B 0,C 180,E1 21930.521,E2 21930.521} C_VEL
LIN {X 0,Y 484.675,Z 575.767,A -85,B 0,C 180,E1 21927.283,E2 21927.283} C_VEL
LIN {X 0,Y 491.407,Z 557.225,A -85,B 0,C 180,E1 21924.558,E2 21924.558} C_VEL
LIN {X 0,Y 498.613,Z 543.248,A -85,B 0,C 180,E1 21922.294,E2 21922.294} C_VEL
LIN {X 0,Y 501.214,Z 539.311,A -85,B 0,C 180,E1 21921.536,E2 21921.536} C_VEL
LIN {X 0,Y 492.979,Z 551.27,A -85,B 0,C 180,E1 21919.989,E2 21919.989} C_VEL
LIN {X 0,Y 485.998,Z 565.215,A -85,B 0,C 180,E1 21918.316,E2 21918.316} C_VEL
LIN {X 0,Y 481.3,Z 579.554,A -85,B 0,C 180,E1 21916.644,E2 21916.644} C_VEL
LIN {X 0,Y 478.822,Z 594.617,A -85,B 0,C 180,E1 21914.895,E2 21914.895} C_VEL
LIN {X 0,Y 478.803,Z 608.074,A -85,B 0,C 180,E1 21913.302,E2 21913.302} C_VEL
LIN {X 0,Y 481.079,Z 621.491,A -85,B 0,C 180,E1 21911.689,E2 21911.689} C_VEL
LIN {X 0,Y 485.242,Z 633.346,A -85,B 0,C 180,E1 21910.233,E2 21910.233} C_VEL
LIN {X 0,Y 491.493,Z 644.617,A -85,B 0,C 180,E1 21908.818,E2 21908.818} C_VEL
LIN {X 0,Y 499.335,Z 654.66,A -85,B 0,C 180,E1 21907.539,E2 21907.539} C_VEL
LIN {X 0,Y 509.66,Z 664.499,A -85,B 0,C 180,E1 21906.264,E2 21906.264} C_VEL
LIN {X 0,Y 516.744,Z 669.987,A -85,B 0,C 180,E1 21905.548,E2 21905.548} C_VEL
LIN {X 0,Y 510.804,Z 680.638,A -85,B 0,C 180,E1 21905.134,E2 21905.134} C_VEL
LIN {X 0,Y 497.845,Z 699.542,A -85,B 0,C 180,E1 21904.498,E2 21904.498} C_VEL
LIN {X 0,Y 488.408,Z 716.01,A -85,B 0,C 180,E1 21903.838,E2 21903.838} C_VEL
LIN {X 0,Y 481.438,Z 731.474,A -85,B 0,C 180,E1 21903.108,E2 21903.108} C_VEL
LIN {X 0,Y 475.786,Z 745.763,A -85,B 0,C 180,E1 21902.416,E2 21902.416} C_VEL
LIN {X 0,Y 472.889,Z 770.51,A -85,B 0,C 180,E1 21902.204,E2 21902.204} C_VEL
LIN {X 0,Y 471.954,Z 805.073,A -85,B 0,C 180,E1 21901.617,E2 21901.617} C_VEL
LIN {X 0,Y 470.941,Z 826.01,A -85,B 0,C 180,E1 21901.04,E2 21901.04} C_VEL
LIN {X 0,Y 469.578,Z 846.478,A -85,B 0,C 180,E1 21900.237,E2 21900.237} C_VEL
LIN {X 0,Y 468.079,Z 865.821,A -85,B 0,C 180,E1 21899.24,E2 21899.24} C_VEL
LIN {X 0,Y 466.369,Z 885.021,A -85,B 0,C 180,E1 21898.004,E2 21898.004} C_VEL
LIN {X 0,Y 464.638,Z 903.003,A -85,B 0,C 180,E1 21896.59,E2 21896.59} C_VEL
LIN {X 0,Y 462.93,Z 920.12,A -85,B 0,C 180,E1 21894.977,E2 21894.977} C_VEL
LIN {X 0,Y 461.334,Z 935.815,A -85,B 0,C 180,E1 21893.228,E2 21893.228} C_VEL
LIN {X 0,Y 459.812,Z 951.436,A -85,B 0,C 180,E1 21891.16,E2 21891.16} C_VEL
LIN {X 0,Y 458.576,Z 965.387,A -85,B 0,C 180,E1 21888.959,E2 21888.959} C_VEL
LIN {X 0,Y 457.563,Z 977.708,A -85,B 0,C 180,E1 21886.635,E2 21886.635} C_VEL
LIN {X 0,Y 456.926,Z 987.365,A -85,B 0,C 180,E1 21884.446,E2 21884.446} C_VEL
LIN {X 0,Y 456.434,Z 997.439,A -85,B 0,C 180,E1 21881.709,E2 21881.709} C_VEL
LIN {X 0,Y 456.185,Z 1004.243,A -85,B 0,C 180,E1 21879.462,E2 21879.462} C_VEL
LIN {X 0,Y 456.05,Z 1009.104,A -85,B 0,C 180,E1 21877.433,E2 21877.433} C_VEL
LIN {X 0,Y 455.997,Z 1013.486,A -85,B 0,C 180,E1 21874.906,E2 21874.906} C_VEL
LIN {X 0,Y 455.983,Z 1015.796,A -85,B 0,C 180,E1 21872.64,E2 21872.64} C_VEL
LIN {X 0,Y 455.972,Z 1016.749,A -85,B 0,C 180,E1 21870.503,E2 21870.503} C_VEL
LIN {X 0,Y 455.978,Z 1016.201,A -85,B 0,C 180,E1 21867.864,E2 21867.864} C_VEL
LIN {X 0,Y 455.982,Z 1014.327,A -85,B 0,C 180,E1 21865.725,E2 21865.725} C_VEL
LIN {X 0,Y 456.016,Z 1011.232,A -85,B 0,C 180,E1 21863.58,E2 21863.58} C_VEL
LIN {X 0,Y 456.121,Z 1005.905,A -85,B 0,C 180,E1 21861.047,E2 21861.047} C_VEL
LIN {X 0,Y 456.321,Z 999.801,A -85,B 0,C 180,E1 21858.883,E2 21858.883} C_VEL
LIN {X 0,Y 456.66,Z 992.274,A -85,B 0,C 180,E1 21856.71,E2 21856.71} C_VEL
LIN {X 0,Y 457.336,Z 980.719,A -85,B 0,C 180,E1 21854.011,E2 21854.011} C_VEL
LIN {X 0,Y 458.222,Z 968.816,A -85,B 0,C 180,E1 21851.656,E2 21851.656} C_VEL
LIN {X 0,Y 459.357,Z 955.74,A -85,B 0,C 180,E1 21849.486,E2 21849.486} C_VEL
LIN {X 0,Y 460.743,Z 941.445,A -85,B 0,C 180,E1 21847.48,E2 21847.48} C_VEL
LIN {X 0,Y 462.31,Z 925.666,A -85,B 0,C 180,E1 21845.602,E2 21845.602} C_VEL
LIN {X 0,Y 464.102,Z 908.208,A -85,B 0,C 180,E1 21843.86,E2 21843.86} C_VEL
LIN {X 0,Y 465.82,Z 890.344,A -85,B 0,C 180,E1 21842.379,E2 21842.379} C_VEL
LIN {X 0,Y 467.521,Z 871.56,A -85,B 0,C 180,E1 21841.097,E2 21841.097} C_VEL
LIN {X 0,Y 469.033,Z 853.102,A -85,B 0,C 180,E1 21840.078,E2 21840.078} C_VEL
LIN {X 0,Y 470.425,Z 832.848,A -85,B 0,C 180,E1 21839.202,E2 21839.202} C_VEL
LIN {X 0,Y 471.566,Z 812.575,A -85,B 0,C 180,E1 21838.562,E2 21838.562} C_VEL
LIN {X 0,Y 472.293,Z 791.352,A -85,B 0,C 180,E1 21838.117,E2 21838.117} C_VEL
LIN {X 0,Y 473.023,Z 766.977,A -85,B 0,C 180,E1 21837.745,E2 21837.745} C_VEL
LIN {X 0,Y 473.561,Z 761.818,A -85,B 0,C 180,E1 21837.677,E2 21837.677} C_VEL
LIN {X 0,Y 479.309,Z 745.604,A -85,B 0,C 180,E1 21836.799,E2 21836.799} C_VEL
LIN {X 0,Y 488.945,Z 723.093,A -85,B 0,C 180,E1 21835.705,E2 21835.705} C_VEL
LIN {X 0,Y 497.672,Z 706.799,A -85,B 0,C 180,E1 21835.07,E2 21835.07} C_VEL
LIN {X 0,Y 509.741,Z 687.982,A -85,B 0,C 180,E1 21834.491,E2 21834.491} C_VEL
LIN {X 0,Y 514.103,Z 681.452,A -85,B 0,C 180,E1 21834.307,E2 21834.307} C_VEL
LIN {X 0,Y 518.82,Z 672.394,A -85,B 0,C 180,E1 21833.968,E2 21833.968} C_VEL
LIN {X 0,Y 508.894,Z 664.689,A -85,B 0,C 180,E1 21832.724,E2 21832.724} C_VEL
LIN {X 0,Y 499.684,Z 654.89,A -85,B 0,C 180,E1 21831.295,E2 21831.295} C_VEL
LIN {X 0,Y 492.122,Z 643.464,A -85,B 0,C 180,E1 21829.812,E2 21829.812} C_VEL
LIN {X 0,Y 486.671,Z 631.501,A -85,B 0,C 180,E1 21828.403,E2 21828.403} C_VEL
LIN {X 0,Y 482.622,Z 617.214,A -85,B 0,C 180,E1 21826.87,E2 21826.87} C_VEL
LIN {X 0,Y 480.342,Z 601.127,A -85,B 0,C 180,E1 21825.287,E2 21825.287} C_VEL
LIN {X 0,Y 479.951,Z 582.116,A -85,B 0,C 180,E1 21823.595,E2 21823.595} C_VEL
LIN {X 0,Y 484.516,Z 527.597,A -85,B 0,C 180,E1 21819.112,E2 21819.112} C_VEL
LIN {X 0,Y 485.464,Z 516.754,A -85,B 0,C 180,E1 21818.202,E2 21818.202} C_VEL
LIN {X 0,Y 475.659,Z 496.26,A -85,B 0,C 180,E1 21815.02,E2 21815.02} C_VEL
LIN {X 0,Y 467.32,Z 479.48,A -85,B 0,C 180,E1 21812.191,E2 21812.191} C_VEL
LIN {X 0,Y 460.973,Z 466.923,A -85,B 0,C 180,E1 21809.925,E2 21809.925} C_VEL
LIN {X 0,Y 459.079,Z 462.973,A -85,B 0,C 180,E1 21809.2,E2 21809.2} C_VEL
LIN {X 0,Y 457.351,Z 460.015,A -85,B 0,C 180,E1 21808.605,E2 21808.605} C_VEL
LIN {X 0,Y 457.041,Z 458.555,A -85,B 0,C 180,E1 21808.341,E2 21808.341} C_VEL
LIN {X 0,Y 457.072,Z 458.551,A -85,B 0,C 180,E1 21804.697,E2 21804.697} C_VEL
LIN {X 0,Y 457.045,Z 458.556,A -85,B 0,C 180,E1 21801.025,E2 21801.025} C_VEL
LIN {X 0,Y 457.062,Z 458.553,A -85,B 0,C 180,E1 21797.308,E2 21797.308} C_VEL
LIN {X 0,Y 457.065,Z 458.554,A -85,B 0,C 180,E1 21793.666,E2 21793.666} C_VEL
LIN {X 0,Y 457.061,Z 458.556,A -85,B 0,C 180,E1 21789.824,E2 21789.824} C_VEL
LIN {X 0,Y 457.06,Z 458.555,A -85,B 0,C 180,E1 21786.153,E2 21786.153} C_VEL
LIN {X 0,Y 457.025,Z 458.556,A -85,B 0,C 180,E1 21782.382,E2 21782.382} C_VEL
LIN {X 0,Y 457.074,Z 458.549,A -85,B 0,C 180,E1 21778.746,E2 21778.746} C_VEL
LIN {X 0,Y 457.044,Z 458.554,A -85,B 0,C 180,E1 21775.105,E2 21775.105} C_VEL
LIN {X 0,Y 457.071,Z 458.538,A -85,B 0,C 180,E1 21771.445,E2 21771.445} C_VEL
LIN {X 0,Y 457.037,Z 458.544,A -85,B 0,C 180,E1 21767.748,E2 21767.748} C_VEL
LIN {X 0,Y 457.052,Z 458.552,A -85,B 0,C 180,E1 21764,E2 21764} C_VEL
LIN {X 0,Y 457.076,Z 458.547,A -85,B 0,C 180,E1 21760.313,E2 21760.313} C_VEL
LIN {X 0,Y 457.07,Z 458.542,A -85,B 0,C 180,E1 21756.538,E2 21756.538} C_VEL
LIN {X 0,Y 457.06,Z 458.543,A -85,B 0,C 180,E1 21752.915,E2 21752.915} C_VEL
LIN {X 0,Y 457.026,Z 458.547,A -85,B 0,C 180,E1 21749.207,E2 21749.207} C_VEL
LIN {X 0,Y 457.069,Z 458.545,A -85,B 0,C 180,E1 21745.557,E2 21745.557} C_VEL
LIN {X 0,Y 457.054,Z 458.546,A -85,B 0,C 180,E1 21741.909,E2 21741.909} C_VEL
LIN {X 0,Y 457.077,Z 458.548,A -85,B 0,C 180,E1 21738.239,E2 21738.239} C_VEL
LIN {X 0,Y 457.039,Z 458.554,A -85,B 0,C 180,E1 21734.505,E2 21734.505} C_VEL
LIN {X 0,Y 457.075,Z 458.737,A -85,B 0,C 180,E1 21731.889,E2 21731.889} C_VEL
LIN {X 0,Y 458.625,Z 462.373,A -85,B 0,C 180,E1 21731.366,E2 21731.366} C_VEL
LIN {X 0,Y 467.098,Z 482.792,A -85,B 0,C 180,E1 21728.528,E2 21728.528} C_VEL
LIN {X 0,Y 473.129,Z 498.641,A -85,B 0,C 180,E1 21726.577,E2 21726.577} C_VEL
LIN {X 0,Y 474.178,Z 501.412,A -85,B 0,C 180,E1 21726.431,E2 21726.431} C_VEL
LIN {X 0,Y 477.906,Z 522.604,A -85,B 0,C 180,E1 21725.711,E2 21725.711} C_VEL
LIN {X 0,Y 475.826,Z 627.058,A -85,B 0,C 180,E1 21723.999,E2 21723.999} C_VEL
LIN {X 0,Y 474.851,Z 634.747,A -85,B 0,C 180,E1 21723.941,E2 21723.941} C_VEL
LIN {X 0,Y 469.266,Z 655.235,A -85,B 0,C 180,E1 21724.032,E2 21724.032} C_VEL
LIN {X 0,Y 468.504,Z 661.834,A -85,B 0,C 180,E1 21723.975,E2 21723.975} C_VEL
LIN {X 0,Y 466.499,Z 760.03,A -85,B 0,C 180,E1 21722.322,E2 21722.322} C_VEL
LIN {X 0,Y 465.559,Z 780.627,A -85,B 0,C 180,E1 21721.765,E2 21721.765} C_VEL
LIN {X 0,Y 464.276,Z 801.002,A -85,B 0,C 180,E1 21720.977,E2 21720.977} C_VEL
LIN {X 0,Y 462.725,Z 820.429,A -85,B 0,C 180,E1 21719.989,E2 21719.989} C_VEL
LIN {X 0,Y 460.976,Z 839.001,A -85,B 0,C 180,E1 21718.803,E2 21718.803} C_VEL
LIN {X 0,Y 459.079,Z 856.956,A -85,B 0,C 180,E1 21717.398,E2 21717.398} C_VEL
LIN {X 0,Y 457.052,Z 874.453,A -85,B 0,C 180,E1 21715.736,E2 21715.736} C_VEL
LIN {X 0,Y 455.134,Z 890.152,A -85,B 0,C 180,E1 21713.951,E2 21713.951} C_VEL
LIN {X 0,Y 453.395,Z 904.51,A -85,B 0,C 180,E1 21712.017,E2 21712.017} C_VEL
LIN {X 0,Y 451.801,Z 918.049,A -85,B 0,C 180,E1 21709.856,E2 21709.856} C_VEL
LIN {X 0,Y 450.49,Z 930.054,A -85,B 0,C 180,E1 21707.568,E2 21707.568} C_VEL
LIN {X 0,Y 449.496,Z 940.336,A -85,B 0,C 180,E1 21705.217,E2 21705.217} C_VEL
LIN {X 0,Y 448.778,Z 949.207,A -85,B 0,C 180,E1 21702.742,E2 21702.742} C_VEL
LIN {X 0,Y 448.313,Z 956.551,A -85,B 0,C 180,E1 21700.147,E2 21700.147} C_VEL
LIN {X 0,Y 448.077,Z 961.824,A -85,B 0,C 180,E1 21697.694,E2 21697.694} C_VEL
LIN {X 0,Y 447.963,Z 965.765,A -85,B 0,C 180,E1 21695.122,E2 21695.122} C_VEL
LIN {X 0,Y 447.936,Z 968.131,A -85,B 0,C 180,E1 21692.558,E2 21692.558} C_VEL
LIN {X 0,Y 447.937,Z 968.961,A -85,B 0,C 180,E1 21689.999,E2 21689.999} C_VEL
LIN {X 0,Y 447.932,Z 968.178,A -85,B 0,C 180,E1 21687.441,E2 21687.441} C_VEL
LIN {X 0,Y 447.964,Z 965.873,A -85,B 0,C 180,E1 21684.877,E2 21684.877} C_VEL
LIN {X 0,Y 448.079,Z 961.801,A -85,B 0,C 180,E1 21682.205,E2 21682.205} C_VEL
LIN {X 0,Y 448.319,Z 956.439,A -85,B 0,C 180,E1 21679.722,E2 21679.722} C_VEL
LIN {X 0,Y 448.789,Z 949.072,A -85,B 0,C 180,E1 21677.126,E2 21677.126} C_VEL
LIN {X 0,Y 449.564,Z 939.674,A -85,B 0,C 180,E1 21674.52,E2 21674.52} C_VEL
LIN {X 0,Y 450.582,Z 929.231,A -85,B 0,C 180,E1 21672.167,E2 21672.167} C_VEL
LIN {X 0,Y 451.877,Z 917.404,A -85,B 0,C 180,E1 21669.942,E2 21669.942} C_VEL
LIN {X 0,Y 453.443,Z 904.133,A -85,B 0,C 180,E1 21667.838,E2 21667.838} C_VEL
LIN {X 0,Y 455.269,Z 889.01,A -85,B 0,C 180,E1 21665.82,E2 21665.82} C_VEL
LIN {X 0,Y 457.174,Z 873.334,A -85,B 0,C 180,E1 21664.061,E2 21664.061} C_VEL
LIN {X 0,Y 459.092,Z 856.84,A -85,B 0,C 180,E1 21662.501,E2 21662.501} C_VEL
LIN {X 0,Y 461.025,Z 838.594,A -85,B 0,C 180,E1 21661.076,E2 21661.076} C_VEL
LIN {X 0,Y 462.737,Z 820.322,A -85,B 0,C 180,E1 21659.914,E2 21659.914} C_VEL
LIN {X 0,Y 464.265,Z 801.229,A -85,B 0,C 180,E1 21658.943,E2 21658.943} C_VEL
LIN {X 0,Y 465.579,Z 780.352,A -85,B 0,C 180,E1 21658.136,E2 21658.136} C_VEL
LIN {X 0,Y 466.516,Z 759.581,A -85,B 0,C 180,E1 21657.578,E2 21657.578} C_VEL
LIN {X 0,Y 471.179,Z 531.965,A -85,B 0,C 180,E1 21653.774,E2 21653.774} C_VEL
LIN {X 0,Y 462.755,Z 500.804,A -85,B 0,C 180,E1 21652.381,E2 21652.381} C_VEL
LIN {X 0,Y 458.901,Z 487.847,A -85,B 0,C 180,E1 21650.275,E2 21650.275} C_VEL
LIN {X 0,Y 453.615,Z 471.975,A -85,B 0,C 180,E1 21647.409,E2 21647.409} C_VEL
LIN {X 0,Y 449.136,Z 459.541,A -85,B 0,C 180,E1 21645.033,E2 21645.033} C_VEL
LIN {X 0,Y 449.139,Z 459.536,A -85,B 0,C 180,E1 21641.196,E2 21641.196} C_VEL
LIN {X 0,Y 449.129,Z 459.544,A -85,B 0,C 180,E1 21637.428,E2 21637.428} C_VEL
LIN {X 0,Y 449.166,Z 459.773,A -85,B 0,C 180,E1 21637.104,E2 21637.104} C_VEL
LIN {X 0,Y 457.252,Z 481.347,A -85,B 0,C 180,E1 21633.691,E2 21633.691} C_VEL
LIN {X 0,Y 463.862,Z 500.795,A -85,B 0,C 180,E1 21630.829,E2 21630.829} C_VEL
LIN {X 0,Y 461.639,Z 534.164,A -85,B 0,C 180,E1 21627.264,E2 21627.264} C_VEL
LIN {X 0,Y 459.402,Z 569.058,A -85,B 0,C 180,E1 21623.607,E2 21623.607} C_VEL
LIN {X 0,Y 457.364,Z 606.577,A -85,B 0,C 180,E1 21619.741,E2 21619.741} C_VEL
LIN {X 0,Y 456.934,Z 617.106,A -85,B 0,C 180,E1 21618.696,E2 21618.696} C_VEL
LIN {X 0,Y 457.618,Z 623.312,A -85,B 0,C 180,E1 21618.523,E2 21618.523} C_VEL
LIN {X 0,Y 454.429,Z 759.95,A -85,B 0,C 180,E1 21615.751,E2 21615.751} C_VEL
LIN {X 0,Y 454.102,Z 777,A -85,B 0,C 180,E1 21615.157,E2 21615.157} C_VEL
LIN {X 0,Y 453.586,Z 792.629,A -85,B 0,C 180,E1 21614.367,E2 21614.367} C_VEL
LIN {X 0,Y 452.947,Z 807.892,A -85,B 0,C 180,E1 21613.337,E2 21613.337} C_VEL
LIN {X 0,Y 452.22,Z 821.823,A -85,B 0,C 180,E1 21612.125,E2 21612.125} C_VEL
LIN {X 0,Y 451.477,Z 834.739,A -85,B 0,C 180,E1 21610.721,E2 21610.721} C_VEL
LIN {X 0,Y 450.795,Z 846.016,A -85,B 0,C 180,E1 21609.189,E2 21609.189} C_VEL
LIN {X 0,Y 450.172,Z 856.59,A -85,B 0,C 180,E1 21607.402,E2 21607.402} C_VEL
LIN {X 0,Y 449.708,Z 864.877,A -85,B 0,C 180,E1 21605.614,E2 21605.614} C_VEL
LIN {X 0,Y 449.353,Z 872.19,A -85,B 0,C 180,E1 21603.572,E2 21603.572} C_VEL
LIN {X 0,Y 449.135,Z 877.389,A -85,B 0,C 180,E1 21601.531,E2 21601.531} C_VEL
LIN {X 0,Y 449.057,Z 880.824,A -85,B 0,C 180,E1 21599.49,E2 21599.49} C_VEL
LIN {X 0,Y 449.051,Z 882.478,A -85,B 0,C 180,E1 21597.448,E2 21597.448} C_VEL
LIN {X 0,Y 449.149,Z 882.49,A -85,B 0,C 180,E1 21595.404,E2 21595.404} C_VEL
LIN {X 0,Y 449.322,Z 880.763,A -85,B 0,C 180,E1 21593.355,E2 21593.355} C_VEL
LIN {X 0,Y 449.643,Z 877.312,A -85,B 0,C 180,E1 21591.303,E2 21591.303} C_VEL
LIN {X 0,Y 450.069,Z 872.298,A -85,B 0,C 180,E1 21589.375,E2 21589.375} C_VEL
LIN {X 0,Y 450.662,Z 865.442,A -85,B 0,C 180,E1 21587.442,E2 21587.442} C_VEL
LIN {X 0,Y 451.378,Z 857.003,A -85,B 0,C 180,E1 21585.635,E2 21585.635} C_VEL
LIN {X 0,Y 452.214,Z 847.059,A -85,B 0,C 180,E1 21583.956,E2 21583.956} C_VEL
LIN {X 0,Y 453.11,Z 835.361,A -85,B 0,C 180,E1 21582.404,E2 21582.404} C_VEL
LIN {X 0,Y 453.955,Z 823.243,A -85,B 0,C 180,E1 21581.109,E2 21581.109} C_VEL
LIN {X 0,Y 454.72,Z 809.258,A -85,B 0,C 180,E1 21579.939,E2 21579.939} C_VEL
LIN {X 0,Y 455.294,Z 795.122,A -85,B 0,C 180,E1 21579.025,E2 21579.025} C_VEL
LIN {X 0,Y 455.712,Z 778.658,A -85,B 0,C 180,E1 21578.248,E2 21578.248} C_VEL
LIN {X 0,Y 455.855,Z 760.27,A -85,B 0,C 180,E1 21577.687,E2 21577.687} C_VEL
LIN {X 0,Y 458.185,Z 707.619,A -85,B 0,C 180,E1 21576.301,E2 21576.301} C_VEL
LIN {X 0,Y 462.454,Z 641.829,A -85,B 0,C 180,E1 21574.488,E2 21574.488} C_VEL
LIN {X 0,Y 467.254,Z 630.334,A -85,B 0,C 180,E1 21573.503,E2 21573.503} C_VEL
LIN {X 0,Y 472.575,Z 603.448,A -85,B 0,C 180,E1 21570.045,E2 21570.045} C_VEL
LIN {X 0,Y 479.389,Z 579.599,A -85,B 0,C 180,E1 21566.733,E2 21566.733} C_VEL
LIN {X 0,Y 486.461,Z 562.104,A -85,B 0,C 180,E1 21564.079,E2 21564.079} C_VEL
LIN {X 0,Y 493.972,Z 548.935,A -85,B 0,C 180,E1 21561.877,E2 21561.877} C_VEL
LIN {X 0,Y 494.699,Z 547.911,A -85,B 0,C 180,E1 21561.648,E2 21561.648} C_VEL
LIN {X 0,Y 486.334,Z 560.029,A -85,B 0,C 180,E1 21560.073,E2 21560.073} C_VEL
LIN {X 0,Y 479.471,Z 573.753,A -85,B 0,C 180,E1 21558.383,E2 21558.383} C_VEL
LIN {X 0,Y 475.069,Z 587.262,A -85,B 0,C 180,E1 21556.738,E2 21556.738} C_VEL
LIN {X 0,Y 472.78,Z 601.002,A -85,B 0,C 180,E1 21555.061,E2 21555.061} C_VEL
LIN {X 0,Y 472.833,Z 614.292,A -85,B 0,C 180,E1 21553.414,E2 21553.414} C_VEL
LIN {X 0,Y 475.154,Z 627.422,A -85,B 0,C 180,E1 21551.758,E2 21551.758} C_VEL
LIN {X 0,Y 479.448,Z 639.223,A -85,B 0,C 180,E1 21550.247,E2 21550.247} C_VEL
LIN {X 0,Y 485.972,Z 650.644,A -85,B 0,C 180,E1 21548.761,E2 21548.761} C_VEL
LIN {X 0,Y 493.812,Z 660.472,A -85,B 0,C 180,E1 21547.467,E2 21547.467} C_VEL
LIN {X 0,Y 504.103,Z 670.196,A -85,B 0,C 180,E1 21546.171,E2 21546.171} C_VEL
LIN {X 0,Y 507.441,Z 672.826,A -85,B 0,C 180,E1 21545.818,E2 21545.818} C_VEL
LIN {X 0,Y 504.187,Z 678.507,A -85,B 0,C 180,E1 21545.603,E2 21545.603} C_VEL
LIN {X 0,Y 491.143,Z 697.668,A -85,B 0,C 180,E1 21544.965,E2 21544.965} C_VEL
LIN {X 0,Y 481.793,Z 714.015,A -85,B 0,C 180,E1 21544.314,E2 21544.314} C_VEL
LIN {X 0,Y 474.633,Z 729.732,A -85,B 0,C 180,E1 21543.573,E2 21543.573} C_VEL
LIN {X 0,Y 469.546,Z 742.461,A -85,B 0,C 180,E1 21542.956,E2 21542.956} C_VEL
LIN {X 0,Y 466.469,Z 766.217,A -85,B 0,C 180,E1 21542.775,E2 21542.775} C_VEL
LIN {X 0,Y 465.722,Z 782.934,A -85,B 0,C 180,E1 21542.535,E2 21542.535} C_VEL
LIN {X 0,Y 464.955,Z 808.689,A -85,B 0,C 180,E1 21542.039,E2 21542.039} C_VEL
LIN {X 0,Y 463.773,Z 829.443,A -85,B 0,C 180,E1 21541.418,E2 21541.418} C_VEL
LIN {X 0,Y 462.4,Z 848.812,A -85,B 0,C 180,E1 21540.616,E2 21540.616} C_VEL
LIN {X 0,Y 460.783,Z 868.102,A -85,B 0,C 180,E1 21539.582,E2 21539.582} C_VEL
LIN {X 0,Y 458.92,Z 887.355,A -85,B 0,C 180,E1 21538.287,E2 21538.287} C_VEL
LIN {X 0,Y 457.079,Z 904.909,A -85,B 0,C 180,E1 21536.848,E2 21536.848} C_VEL
LIN {X 0,Y 455.263,Z 921.749,A -85,B 0,C 180,E1 21535.198,E2 21535.198} C_VEL
LIN {X 0,Y 453.493,Z 937.948,A -85,B 0,C 180,E1 21533.314,E2 21533.314} C_VEL
LIN {X 0,Y 451.943,Z 952.744,A -85,B 0,C 180,E1 21531.275,E2 21531.275} C_VEL
LIN {X 0,Y 450.668,Z 966.246,A -85,B 0,C 180,E1 21529.069,E2 21529.069} C_VEL
LIN {X 0,Y 449.645,Z 977.937,A -85,B 0,C 180,E1 21526.803,E2 21526.803} C_VEL
LIN {X 0,Y 448.933,Z 988.021,A -85,B 0,C 180,E1 21524.445,E2 21524.445} C_VEL
LIN {X 0,Y 448.476,Z 996.291,A -85,B 0,C 180,E1 21522.098,E2 21522.098} C_VEL
LIN {X 0,Y 448.208,Z 1003.596,A -85,B 0,C 180,E1 21519.502,E2 21519.502} C_VEL
LIN {X 0,Y 448.099,Z 1009.875,A -85,B 0,C 180,E1 21516.535,E2 21516.535} C_VEL
LIN {X 0,Y 448.063,Z 1013.091,A -85,B 0,C 180,E1 21514.352,E2 21514.352} C_VEL
LIN {X 0,Y 448.055,Z 1015.142,A -85,B 0,C 180,E1 21512.047,E2 21512.047} C_VEL
LIN {X 0,Y 448.043,Z 1015.68,A -85,B 0,C 180,E1 21509.489,E2 21509.489} C_VEL
LIN {X 0,Y 448.042,Z 1014.782,A -85,B 0,C 180,E1 21507.315,E2 21507.315} C_VEL
LIN {X 0,Y 448.04,Z 1012.516,A -85,B 0,C 180,E1 21505.008,E2 21505.008} C_VEL
LIN {X 0,Y 448.078,Z 1008.221,A -85,B 0,C 180,E1 21502.435,E2 21502.435} C_VEL
LIN {X 0,Y 448.216,Z 1003.116,A -85,B 0,C 180,E1 21500.24,E2 21500.24} C_VEL
LIN {X 0,Y 448.507,Z 995.053,A -85,B 0,C 180,E1 21497.512,E2 21497.512} C_VEL
LIN {X 0,Y 449.045,Z 985.923,A -85,B 0,C 180,E1 21495.032,E2 21495.032} C_VEL
LIN {X 0,Y 449.817,Z 975.355,A -85,B 0,C 180,E1 21492.672,E2 21492.672} C_VEL
LIN {X 0,Y 450.874,Z 963.415,A -85,B 0,C 180,E1 21490.437,E2 21490.437} C_VEL
LIN {X 0,Y 452.194,Z 950.126,A -85,B 0,C 180,E1 21488.331,E2 21488.331} C_VEL
LIN {X 0,Y 453.795,Z 934.871,A -85,B 0,C 180,E1 21486.291,E2 21486.291} C_VEL
LIN {X 0,Y 455.649,Z 917.887,A -85,B 0,C 180,E1 21484.388,E2 21484.388} C_VEL
LIN {X 0,Y 457.514,Z 900.397,A -85,B 0,C 180,E1 21482.753,E2 21482.753} C_VEL
LIN {X 0,Y 459.295,Z 882.829,A -85,B 0,C 180,E1 21481.385,E2 21481.385} C_VEL
LIN {X 0,Y 461.114,Z 863.468,A -85,B 0,C 180,E1 21480.151,E2 21480.151} C_VEL
LIN {X 0,Y 462.701,Z 843.911,A -85,B 0,C 180,E1 21479.158,E2 21479.158} C_VEL
LIN {X 0,Y 464.087,Z 824,A -85,B 0,C 180,E1 21478.39,E2 21478.39} C_VEL
LIN {X 0,Y 465.145,Z 803.107,A -85,B 0,C 180,E1 21477.821,E2 21477.821} C_VEL
LIN {X 0,Y 466.176,Z 768.133,A -85,B 0,C 180,E1 21477.238,E2 21477.238} C_VEL
LIN {X 0,Y 467.038,Z 759.804,A -85,B 0,C 180,E1 21477.133,E2 21477.133} C_VEL
LIN {X 0,Y 472.385,Z 744.91,A -85,B 0,C 180,E1 21476.321,E2 21476.321} C_VEL
LIN {X 0,Y 482.408,Z 721.682,A -85,B 0,C 180,E1 21475.187,E2 21475.187} C_VEL
LIN {X 0,Y 491.174,Z 705.504,A -85,B 0,C 180,E1 21474.539,E2 21474.539} C_VEL
LIN {X 0,Y 503.304,Z 686.518,A -85,B 0,C 180,E1 21473.953,E2 21473.953} C_VEL
LIN {X 0,Y 508.471,Z 678.665,A -85,B 0,C 180,E1 21473.728,E2 21473.728} C_VEL
LIN {X 0,Y 509.799,Z 675.735,A -85,B 0,C 180,E1 21473.605,E2 21473.605} C_VEL
LIN {X 0,Y 499.675,Z 666.921,A -85,B 0,C 180,E1 21472.223,E2 21472.223} C_VEL
LIN {X 0,Y 491.347,Z 657.067,A -85,B 0,C 180,E1 21470.833,E2 21470.833} C_VEL
LIN {X 0,Y 484.081,Z 645.01,A -85,B 0,C 180,E1 21469.291,E2 21469.291} C_VEL
LIN {X 0,Y 478.962,Z 632.409,A -85,B 0,C 180,E1 21467.823,E2 21467.823} C_VEL
LIN {X 0,Y 475.328,Z 617.814,A -85,B 0,C 180,E1 21466.266,E2 21466.266} C_VEL
LIN {X 0,Y 473.42,Z 601.685,A -85,B 0,C 180,E1 21464.692,E2 21464.692} C_VEL
LIN {X 0,Y 473.407,Z 581.289,A -85,B 0,C 180,E1 21462.873,E2 21462.873} C_VEL
LIN {X 0,Y 477.892,Z 532.125,A -85,B 0,C 180,E1 21458.8,E2 21458.8} C_VEL
LIN {X 0,Y 479.025,Z 520.874,A -85,B 0,C 180,E1 21457.854,E2 21457.854} C_VEL
LIN {X 0,Y 470.088,Z 501.973,A -85,B 0,C 180,E1 21454.9,E2 21454.9} C_VEL
LIN {X 0,Y 461.421,Z 484.466,A -85,B 0,C 180,E1 21451.919,E2 21451.919} C_VEL
LIN {X 0,Y 454.727,Z 471.326,A -85,B 0,C 180,E1 21449.507,E2 21449.507} C_VEL
LIN {X 0,Y 453.105,Z 468.073,A -85,B 0,C 180,E1 21448.899,E2 21448.899} C_VEL
LIN {X 0,Y 450.872,Z 463.619,A -85,B 0,C 180,E1 21448.043,E2 21448.043} C_VEL
LIN {X 0,Y 449.281,Z 460.516,A -85,B 0,C 180,E1 21447.43,E2 21447.43} C_VEL
LIN {X 0,Y 449.094,Z 459.544,A -85,B 0,C 180,E1 21447.24,E2 21447.24} C_VEL
LIN {X 0,Y 449.139,Z 459.541,A -85,B 0,C 180,E1 21443.622,E2 21443.622} C_VEL
LIN {X 0,Y 449.104,Z 459.543,A -85,B 0,C 180,E1 21440.032,E2 21440.032} C_VEL
LIN {X 0,Y 449.133,Z 459.541,A -85,B 0,C 180,E1 21436.366,E2 21436.366} C_VEL
LIN {X 0,Y 449.106,Z 459.545,A -85,B 0,C 180,E1 21432.733,E2 21432.733} C_VEL
LIN {X 0,Y 449.117,Z 459.541,A -85,B 0,C 180,E1 21428.836,E2 21428.836} C_VEL
LIN {X 0,Y 449.137,Z 459.539,A -85,B 0,C 180,E1 21425.109,E2 21425.109} C_VEL
LIN {X 0,Y 449.14,Z 459.537,A -85,B 0,C 180,E1 21421.148,E2 21421.148} C_VEL
LIN {X 0,Y 449.115,Z 459.541,A -85,B 0,C 180,E1 21417.448,E2 21417.448} C_VEL
LIN {X 0,Y 449.095,Z 459.542,A -85,B 0,C 180,E1 21413.608,E2 21413.608} C_VEL
LIN {X 0,Y 449.131,Z 459.539,A -85,B 0,C 180,E1 21410,E2 21410} C_VEL
LIN {X 0,Y 449.114,Z 459.529,A -85,B 0,C 180,E1 21406.35,E2 21406.35} C_VEL
LIN {X 0,Y 449.135,Z 459.529,A -85,B 0,C 180,E1 21402.751,E2 21402.751} C_VEL
LIN {X 0,Y 449.091,Z 459.544,A -85,B 0,C 180,E1 21399.131,E2 21399.131} C_VEL
LIN {X 0,Y 449.117,Z 459.542,A -85,B 0,C 180,E1 21395.273,E2 21395.273} C_VEL
LIN {X 0,Y 449.13,Z 459.54,A -85,B 0,C 180,E1 21391.549,E2 21391.549} C_VEL
LIN {X 0,Y 449.127,Z 459.542,A -85,B 0,C 180,E1 21387.774,E2 21387.774} C_VEL
LIN {X 0,Y 449.123,Z 459.542,A -85,B 0,C 180,E1 21384.129,E2 21384.129} C_VEL
LIN {X 0,Y 449.098,Z 459.546,A -85,B 0,C 180,E1 21380.382,E2 21380.382} C_VEL
LIN {X 0,Y 449.133,Z 459.536,A -85,B 0,C 180,E1 21376.711,E2 21376.711} C_VEL
LIN {X 0,Y 449.108,Z 459.547,A -85,B 0,C 180,E1 21373.094,E2 21373.094} C_VEL
LIN {X 0,Y 449.124,Z 459.807,A -85,B 0,C 180,E1 21372.681,E2 21372.681} C_VEL
LIN {X 0,Y 450.579,Z 463.284,A -85,B 0,C 180,E1 21372.169,E2 21372.169} C_VEL
LIN {X 0,Y 458.317,Z 481.253,A -85,B 0,C 180,E1 21369.569,E2 21369.569} C_VEL
LIN {X 0,Y 465.232,Z 498.883,A -85,B 0,C 180,E1 21367.305,E2 21367.305} C_VEL
LIN {X 0,Y 468.082,Z 504.73,A -85,B 0,C 180,E1 21366.926,E2 21366.926} C_VEL
LIN {X 0,Y 471.408,Z 524.122,A -85,B 0,C 180,E1 21366.258,E2 21366.258} C_VEL
LIN {X 0,Y 468.504,Z 661.834,A -85,B 0,C 180,E1 21363.975,E2 21363.975} C_VEL
LIN {X 0,Y 467.523,Z 669.523,A -85,B 0,C 180,E1 21363.917,E2 21363.917} C_VEL
LIN {X 0,Y 461.951,Z 690.011,A -85,B 0,C 180,E1 21364.008,E2 21364.008} C_VEL
LIN {X 0,Y 461.18,Z 696.611,A -85,B 0,C 180,E1 21363.951,E2 21363.951} C_VEL
LIN {X 0,Y 459.737,Z 761.13,A -85,B 0,C 180,E1 21362.839,E2 21362.839} C_VEL
LIN {X 0,Y 458.747,Z 781.478,A -85,B 0,C 180,E1 21362.274,E2 21362.274} C_VEL
LIN {X 0,Y 457.422,Z 801.375,A -85,B 0,C 180,E1 21361.494,E2 21361.494} C_VEL
LIN {X 0,Y 455.847,Z 820.263,A -85,B 0,C 180,E1 21360.526,E2 21360.526} C_VEL
LIN {X 0,Y 454.013,Z 838.755,A -85,B 0,C 180,E1 21359.34,E2 21359.34} C_VEL
LIN {X 0,Y 451.971,Z 857.029,A -85,B 0,C 180,E1 21357.896,E2 21357.896} C_VEL
LIN {X 0,Y 449.852,Z 874.207,A -85,B 0,C 180,E1 21356.25,E2 21356.25} C_VEL
LIN {X 0,Y 447.836,Z 889.799,A -85,B 0,C 180,E1 21354.465,E2 21354.465} C_VEL
LIN {X 0,Y 445.997,Z 904.058,A -85,B 0,C 180,E1 21352.535,E2 21352.535} C_VEL
LIN {X 0,Y 444.312,Z 917.324,A -85,B 0,C 180,E1 21350.413,E2 21350.413} C_VEL
LIN {X 0,Y 442.88,Z 929.428,A -85,B 0,C 180,E1 21348.109,E2 21348.109} C_VEL
LIN {X 0,Y 441.781,Z 939.74,A -85,B 0,C 180,E1 21345.758,E2 21345.758} C_VEL
LIN {X 0,Y 440.928,Z 949.195,A -85,B 0,C 180,E1 21343.106,E2 21343.106} C_VEL
LIN {X 0,Y 440.393,Z 956.625,A -85,B 0,C 180,E1 21340.464,E2 21340.464} C_VEL
LIN {X 0,Y 440.122,Z 962.104,A -85,B 0,C 180,E1 21337.905,E2 21337.905} C_VEL
LIN {X 0,Y 439.981,Z 966.178,A -85,B 0,C 180,E1 21335.215,E2 21335.215} C_VEL
LIN {X 0,Y 439.948,Z 968.543,A -85,B 0,C 180,E1 21332.604,E2 21332.604} C_VEL
LIN {X 0,Y 439.948,Z 969.373,A -85,B 0,C 180,E1 21329.999,E2 21329.999} C_VEL
LIN {X 0,Y 439.943,Z 968.589,A -85,B 0,C 180,E1 21327.394,E2 21327.394} C_VEL
LIN {X 0,Y 439.981,Z 966.284,A -85,B 0,C 180,E1 21324.784,E2 21324.784} C_VEL
LIN {X 0,Y 440.114,Z 962.286,A -85,B 0,C 180,E1 21322.103,E2 21322.103} C_VEL
LIN {X 0,Y 440.382,Z 956.85,A -85,B 0,C 180,E1 21319.534,E2 21319.534} C_VEL
LIN {X 0,Y 440.906,Z 949.482,A -85,B 0,C 180,E1 21316.892,E2 21316.892} C_VEL
LIN {X 0,Y 441.747,Z 940.083,A -85,B 0,C 180,E1 21314.239,E2 21314.239} C_VEL
LIN {X 0,Y 442.855,Z 929.636,A -85,B 0,C 180,E1 21311.845,E2 21311.845} C_VEL
LIN {X 0,Y 444.252,Z 917.805,A -85,B 0,C 180,E1 21309.582,E2 21309.582} C_VEL
LIN {X 0,Y 445.927,Z 904.594,A -85,B 0,C 180,E1 21307.454,E2 21307.454} C_VEL
LIN {X 0,Y 447.818,Z 889.946,A -85,B 0,C 180,E1 21305.462,E2 21305.462} C_VEL
LIN {X 0,Y 449.835,Z 874.375,A -85,B 0,C 180,E1 21303.676,E2 21303.676} C_VEL
LIN {X 0,Y 451.95,Z 857.224,A -85,B 0,C 180,E1 21302.029,E2 21302.029} C_VEL
LIN {X 0,Y 453.995,Z 838.973,A -85,B 0,C 180,E1 21300.585,E2 21300.585} C_VEL
LIN {X 0,Y 455.808,Z 820.689,A -85,B 0,C 180,E1 21299.408,E2 21299.408} C_VEL
LIN {X 0,Y 457.408,Z 801.66,A -85,B 0,C 180,E1 21298.428,E2 21298.428} C_VEL
LIN {X 0,Y 458.795,Z 780.795,A -85,B 0,C 180,E1 21297.612,E2 21297.612} C_VEL
LIN {X 0,Y 459.777,Z 760.034,A -85,B 0,C 180,E1 21297.047,E2 21297.047} C_VEL
LIN {X 0,Y 464.712,Z 535.117,A -85,B 0,C 180,E1 21293.244,E2 21293.244} C_VEL
LIN {X 0,Y 464.286,Z 532.126,A -85,B 0,C 180,E1 21293.147,E2 21293.147} C_VEL
LIN {X 0,Y 456.71,Z 504.504,A -85,B 0,C 180,E1 21291.885,E2 21291.885} C_VEL
LIN {X 0,Y 455.095,Z 501.389,A -85,B 0,C 180,E1 21291.66,E2 21291.66} C_VEL
LIN {X 0,Y 449.898,Z 484.964,A -85,B 0,C 180,E1 21288.864,E2 21288.864} C_VEL
LIN {X 0,Y 444.916,Z 470.505,A -85,B 0,C 180,E1 21286.169,E2 21286.169} C_VEL
LIN {X 0,Y 441.183,Z 460.524,A -85,B 0,C 180,E1 21284.18,E2 21284.18} C_VEL
LIN {X 0,Y 441.202,Z 460.528,A -85,B 0,C 180,E1 21280.402,E2 21280.402} C_VEL
LIN {X 0,Y 441.197,Z 460.603,A -85,B 0,C 180,E1 21277.86,E2 21277.86} C_VEL
LIN {X 0,Y 449.165,Z 481.774,A -85,B 0,C 180,E1 21274.431,E2 21274.431} C_VEL
LIN {X 0,Y 455.805,Z 500.882,A -85,B 0,C 180,E1 21271.545,E2 21271.545} C_VEL
LIN {X 0,Y 456.687,Z 504.568,A -85,B 0,C 180,E1 21271.038,E2 21271.038} C_VEL
LIN {X 0,Y 454.329,Z 538.495,A -85,B 0,C 180,E1 21267.384,E2 21267.384} C_VEL
LIN {X 0,Y 451.977,Z 573.62,A -85,B 0,C 180,E1 21263.672,E2 21263.672} C_VEL
LIN {X 0,Y 449.842,Z 610.72,A -85,B 0,C 180,E1 21259.814,E2 21259.814} C_VEL
LIN {X 0,Y 449.567,Z 618.188,A -85,B 0,C 180,E1 21259.08,E2 21259.08} C_VEL
LIN {X 0,Y 450.249,Z 624.306,A -85,B 0,C 180,E1 21258.906,E2 21258.906} C_VEL
LIN {X 0,Y 446.811,Z 760.779,A -85,B 0,C 180,E1 21256.048,E2 21256.048} C_VEL
LIN {X 0,Y 446.471,Z 777.512,A -85,B 0,C 180,E1 21255.456,E2 21255.456} C_VEL
LIN {X 0,Y 445.951,Z 792.875,A -85,B 0,C 180,E1 21254.676,E2 21254.676} C_VEL
LIN {X 0,Y 445.278,Z 808.176,A -85,B 0,C 180,E1 21253.638,E2 21253.638} C_VEL
LIN {X 0,Y 444.558,Z 821.663,A -85,B 0,C 180,E1 21252.469,E2 21252.469} C_VEL
LIN {X 0,Y 443.731,Z 835.34,A -85,B 0,C 180,E1 21250.977,E2 21250.977} C_VEL
LIN {X 0,Y 443.039,Z 846.341,A -85,B 0,C 180,E1 21249.483,E2 21249.483} C_VEL
LIN {X 0,Y 442.366,Z 857.075,A -85,B 0,C 180,E1 21247.664,E2 21247.664} C_VEL
LIN {X 0,Y 441.866,Z 865.563,A -85,B 0,C 180,E1 21245.845,E2 21245.845} C_VEL
LIN {X 0,Y 441.481,Z 873.016,A -85,B 0,C 180,E1 21243.766,E2 21243.766} C_VEL
LIN {X 0,Y 441.254,Z 878.109,A -85,B 0,C 180,E1 21241.818,E2 21241.818} C_VEL
LIN {X 0,Y 441.156,Z 881.932,A -85,B 0,C 180,E1 21239.611,E2 21239.611} C_VEL
LIN {X 0,Y 441.153,Z 883.73,A -85,B 0,C 180,E1 21237.532,E2 21237.532} C_VEL
LIN {X 0,Y 441.268,Z 883.815,A -85,B 0,C 180,E1 21235.321,E2 21235.321} C_VEL
LIN {X 0,Y 441.468,Z 882.096,A -85,B 0,C 180,E1 21233.237,E2 21233.237} C_VEL
LIN {X 0,Y 441.827,Z 878.674,A -85,B 0,C 180,E1 21231.148,E2 21231.148} C_VEL
LIN {X 0,Y 442.303,Z 873.679,A -85,B 0,C 180,E1 21229.186,E2 21229.186} C_VEL
LIN {X 0,Y 442.973,Z 866.722,A -85,B 0,C 180,E1 21227.188,E2 21227.188} C_VEL
LIN {X 0,Y 443.737,Z 858.402,A -85,B 0,C 180,E1 21225.383,E2 21225.383} C_VEL
LIN {X 0,Y 444.653,Z 848.509,A -85,B 0,C 180,E1 21223.676,E2 21223.676} C_VEL
LIN {X 0,Y 445.629,Z 836.881,A -85,B 0,C 180,E1 21222.098,E2 21222.098} C_VEL
LIN {X 0,Y 446.529,Z 824.753,A -85,B 0,C 180,E1 21220.782,E2 21220.782} C_VEL
LIN {X 0,Y 447.415,Z 810.043,A -85,B 0,C 180,E1 21219.529,E2 21219.529} C_VEL
LIN {X 0,Y 448.026,Z 795.695,A -85,B 0,C 180,E1 21218.6,E2 21218.6} C_VEL
LIN {X 0,Y 448.453,Z 780.227,A -85,B 0,C 180,E1 21217.86,E2 21217.86} C_VEL
LIN {X 0,Y 448.718,Z 758.156,A -85,B 0,C 180,E1 21217.175,E2 21217.175} C_VEL
LIN {X 0,Y 452.246,Z 694.715,A -85,B 0,C 180,E1 21215.392,E2 21215.392} C_VEL
LIN {X 0,Y 456.075,Z 644.503,A -85,B 0,C 180,E1 21213.924,E2 21213.924} C_VEL
LIN {X 0,Y 461.205,Z 632.761,A -85,B 0,C 180,E1 21212.918,E2 21212.918} C_VEL
LIN {X 0,Y 466.882,Z 606.85,A -85,B 0,C 180,E1 21209.499,E2 21209.499} C_VEL
LIN {X 0,Y 473.62,Z 585.24,A -85,B 0,C 180,E1 21206.42,E2 21206.42} C_VEL
LIN {X 0,Y 481.264,Z 567.886,A -85,B 0,C 180,E1 21203.717,E2 21203.717} C_VEL
LIN {X 0,Y 488.18,Z 556.518,A -85,B 0,C 180,E1 21201.764,E2 21201.764} C_VEL
LIN {X 0,Y 479.511,Z 569.132,A -85,B 0,C 180,E1 21200.117,E2 21200.117} C_VEL
LIN {X 0,Y 472.996,Z 582.247,A -85,B 0,C 180,E1 21198.446,E2 21198.446} C_VEL
LIN {X 0,Y 468.826,Z 595.174,A -85,B 0,C 180,E1 21196.797,E2 21196.797} C_VEL
LIN {X 0,Y 466.728,Z 608.586,A -85,B 0,C 180,E1 21195.075,E2 21195.075} C_VEL
LIN {X 0,Y 466.979,Z 621.292,A -85,B 0,C 180,E1 21193.418,E2 21193.418} C_VEL
LIN {X 0,Y 469.513,Z 634.184,A -85,B 0,C 180,E1 21191.72,E2 21191.72} C_VEL
LIN {X 0,Y 474.122,Z 646.006,A -85,B 0,C 180,E1 21190.141,E2 21190.141} C_VEL
LIN {X 0,Y 481.2,Z 657.704,A -85,B 0,C 180,E1 21188.562,E2 21188.562} C_VEL
LIN {X 0,Y 490.261,Z 668.33,A -85,B 0,C 180,E1 21187.116,E2 21187.116} C_VEL
LIN {X 0,Y 498.168,Z 675.717,A -85,B 0,C 180,E1 21186.115,E2 21186.115} C_VEL
LIN {X 0,Y 485.059,Z 695.017,A -85,B 0,C 180,E1 21185.49,E2 21185.49} C_VEL
LIN {X 0,Y 475.372,Z 711.845,A -85,B 0,C 180,E1 21184.824,E2 21184.824} C_VEL
LIN {X 0,Y 467.835,Z 728.199,A -85,B 0,C 180,E1 21184.053,E2 21184.053} C_VEL
LIN {X 0,Y 463.313,Z 739.503,A -85,B 0,C 180,E1 21183.507,E2 21183.507} C_VEL
LIN {X 0,Y 460.319,Z 760.771,A -85,B 0,C 180,E1 21183.364,E2 21183.364} C_VEL
LIN {X 0,Y 459.071,Z 777.859,A -85,B 0,C 180,E1 21183.154,E2 21183.154} C_VEL
LIN {X 0,Y 458.265,Z 806.15,A -85,B 0,C 180,E1 21182.628,E2 21182.628} C_VEL
LIN {X 0,Y 457.123,Z 826.501,A -85,B 0,C 180,E1 21182.039,E2 21182.039} C_VEL
LIN {X 0,Y 455.63,Z 846.29,A -85,B 0,C 180,E1 21181.239,E2 21181.239} C_VEL
LIN {X 0,Y 453.937,Z 865.458,A -85,B 0,C 180,E1 21180.22,E2 21180.22} C_VEL
LIN {X 0,Y 452.026,Z 884.248,A -85,B 0,C 180,E1 21178.975,E2 21178.975} C_VEL
LIN {X 0,Y 450.039,Z 902.214,A -85,B 0,C 180,E1 21177.525,E2 21177.525} C_VEL
LIN {X 0,Y 448.087,Z 919.319,A -85,B 0,C 180,E1 21175.865,E2 21175.865} C_VEL
LIN {X 0,Y 446.25,Z 934.973,A -85,B 0,C 180,E1 21174.067,E2 21174.067} C_VEL
LIN {X 0,Y 444.58,Z 949.708,A -85,B 0,C 180,E1 21172.061,E2 21172.061} C_VEL
LIN {X 0,Y 443.155,Z 962.994,A -85,B 0,C 180,E1 21169.92,E2 21169.92} C_VEL
LIN {X 0,Y 442.001,Z 974.934,A -85,B 0,C 180,E1 21167.646,E2 21167.646} C_VEL
LIN {X 0,Y 441.151,Z 985.501,A -85,B 0,C 180,E1 21165.244,E2 21165.244} C_VEL
LIN {X 0,Y 440.586,Z 994.631,A -85,B 0,C 180,E1 21162.717,E2 21162.717} C_VEL
LIN {X 0,Y 440.261,Z 1001.921,A -85,B 0,C 180,E1 21160.204,E2 21160.204} C_VEL
LIN {X 0,Y 440.115,Z 1007.683,A -85,B 0,C 180,E1 21157.572,E2 21157.572} C_VEL
LIN {X 0,Y 440.09,Z 1011.504,A -85,B 0,C 180,E1 21155.084,E2 21155.084} C_VEL
LIN {X 0,Y 440.107,Z 1013.911,A -85,B 0,C 180,E1 21152.475,E2 21152.475} C_VEL
LIN {X 0,Y 440.126,Z 1014.684,A -85,B 0,C 180,E1 21149.871,E2 21149.871} C_VEL
LIN {X 0,Y 440.102,Z 1013.771,A -85,B 0,C 180,E1 21147.266,E2 21147.266} C_VEL
LIN {X 0,Y 440.083,Z 1011.339,A -85,B 0,C 180,E1 21144.787,E2 21144.787} C_VEL
LIN {X 0,Y 440.117,Z 1007.165,A -85,B 0,C 180,E1 21142.166,E2 21142.166} C_VEL
LIN {X 0,Y 440.258,Z 1001.581,A -85,B 0,C 180,E1 21139.665,E2 21139.665} C_VEL
LIN {X 0,Y 440.607,Z 993.807,A -85,B 0,C 180,E1 21137.018,E2 21137.018} C_VEL
LIN {X 0,Y 441.207,Z 984.455,A -85,B 0,C 180,E1 21134.49,E2 21134.49} C_VEL
LIN {X 0,Y 442.084,Z 973.645,A -85,B 0,C 180,E1 21132.087,E2 21132.087} C_VEL
LIN {X 0,Y 443.292,Z 961.176,A -85,B 0,C 180,E1 21129.767,E2 21129.767} C_VEL
LIN {X 0,Y 444.833,Z 946.897,A -85,B 0,C 180,E1 21127.536,E2 21127.536} C_VEL
LIN {X 0,Y 446.582,Z 931.675,A -85,B 0,C 180,E1 21125.532,E2 21125.532} C_VEL
LIN {X 0,Y 448.479,Z 915.523,A -85,B 0,C 180,E1 21123.734,E2 21123.734} C_VEL
LIN {X 0,Y 450.5,Z 897.735,A -85,B 0,C 180,E1 21122.077,E2 21122.077} C_VEL
LIN {X 0,Y 452.561,Z 878.81,A -85,B 0,C 180,E1 21120.629,E2 21120.629} C_VEL
LIN {X 0,Y 454.393,Z 859.778,A -85,B 0,C 180,E1 21119.45,E2 21119.45} C_VEL
LIN {X 0,Y 456.017,Z 840.581,A -85,B 0,C 180,E1 21118.508,E2 21118.508} C_VEL
LIN {X 0,Y 457.46,Z 819.624,A -85,B 0,C 180,E1 21117.735,E2 21117.735} C_VEL
LIN {X 0,Y 458.521,Z 798.124,A -85,B 0,C 180,E1 21117.196,E2 21117.196} C_VEL
LIN {X 0,Y 459.471,Z 767.875,A -85,B 0,C 180,E1 21116.698,E2 21116.698} C_VEL
LIN {X 0,Y 460.553,Z 757.751,A -85,B 0,C 180,E1 21116.573,E2 21116.573} C_VEL
LIN {X 0,Y 465.861,Z 743.361,A -85,B 0,C 180,E1 21115.784,E2 21115.784} C_VEL
LIN {X 0,Y 476.028,Z 720.043,A -85,B 0,C 180,E1 21114.644,E2 21114.644} C_VEL
LIN {X 0,Y 485.266,Z 703.169,A -85,B 0,C 180,E1 21113.968,E2 21113.968} C_VEL
LIN {X 0,Y 497.144,Z 684.725,A -85,B 0,C 180,E1 21113.394,E2 21113.394} C_VEL
LIN {X 0,Y 501.007,Z 678.977,A -85,B 0,C 180,E1 21113.236,E2 21113.236} C_VEL
LIN {X 0,Y 490.775,Z 669.106,A -85,B 0,C 180,E1 21111.733,E2 21111.733} C_VEL
LIN {X 0,Y 483.091,Z 659.062,A -85,B 0,C 180,E1 21110.347,E2 21110.347} C_VEL
LIN {X 0,Y 476.121,Z 646.369,A -85,B 0,C 180,E1 21108.747,E2 21108.747} C_VEL
LIN {X 0,Y 471.143,Z 632.529,A -85,B 0,C 180,E1 21107.157,E2 21107.157} C_VEL
LIN {X 0,Y 467.838,Z 616.724,A -85,B 0,C 180,E1 21105.494,E2 21105.494} C_VEL
LIN {X 0,Y 466.491,Z 599.979,A -85,B 0,C 180,E1 21103.875,E2 21103.875} C_VEL
LIN {X 0,Y 467.107,Z 578.121,A -85,B 0,C 180,E1 21101.942,E2 21101.942} C_VEL
LIN {X 0,Y 471.375,Z 535.645,A -85,B 0,C 180,E1 21098.394,E2 21098.394} C_VEL
LIN {X 0,Y 472.455,Z 524.589,A -85,B 0,C 180,E1 21097.446,E2 21097.446} C_VEL
LIN {X 0,Y 463.424,Z 505.551,A -85,B 0,C 180,E1 21094.421,E2 21094.421} C_VEL
LIN {X 0,Y 454.371,Z 486.957,A -85,B 0,C 180,E1 21091.213,E2 21091.213} C_VEL
LIN {X 0,Y 447.533,Z 473.628,A -85,B 0,C 180,E1 21088.708,E2 21088.708} C_VEL
LIN {X 0,Y 443.067,Z 464.805,A -85,B 0,C 180,E1 21086.974,E2 21086.974} C_VEL
LIN {X 0,Y 441.458,Z 461.818,A -85,B 0,C 180,E1 21086.354,E2 21086.354} C_VEL
LIN {X 0,Y 441.198,Z 460.527,A -85,B 0,C 180,E1 21086.117,E2 21086.117} C_VEL
LIN {X 0,Y 441.174,Z 460.533,A -85,B 0,C 180,E1 21082.38,E2 21082.38} C_VEL
LIN {X 0,Y 441.16,Z 460.533,A -85,B 0,C 180,E1 21078.5,E2 21078.5} C_VEL
LIN {X 0,Y 441.2,Z 460.529,A -85,B 0,C 180,E1 21074.838,E2 21074.838} C_VEL
LIN {X 0,Y 441.167,Z 460.533,A -85,B 0,C 180,E1 21071.087,E2 21071.087} C_VEL
LIN {X 0,Y 441.199,Z 460.527,A -85,B 0,C 180,E1 21067.422,E2 21067.422} C_VEL
LIN {X 0,Y 441.149,Z 460.535,A -85,B 0,C 180,E1 21063.768,E2 21063.768} C_VEL
LIN {X 0,Y 441.187,Z 460.529,A -85,B 0,C 180,E1 21060,E2 21060} C_VEL
LIN {X 0,Y 441.178,Z 460.529,A -85,B 0,C 180,E1 21056.362,E2 21056.362} C_VEL
LIN {X 0,Y 441.181,Z 460.513,A -85,B 0,C 180,E1 21052.447,E2 21052.447} C_VEL
LIN {X 0,Y 441.189,Z 460.528,A -85,B 0,C 180,E1 21048.761,E2 21048.761} C_VEL
LIN {X 0,Y 441.19,Z 460.529,A -85,B 0,C 180,E1 21044.889,E2 21044.889} C_VEL
LIN {X 0,Y 441.183,Z 460.519,A -85,B 0,C 180,E1 21041.227,E2 21041.227} C_VEL
LIN {X 0,Y 441.146,Z 460.519,A -85,B 0,C 180,E1 21037.478,E2 21037.478} C_VEL
LIN {X 0,Y 441.193,Z 460.523,A -85,B 0,C 180,E1 21033.773,E2 21033.773} C_VEL
LIN {X 0,Y 441.187,Z 460.528,A -85,B 0,C 180,E1 21030.093,E2 21030.093} C_VEL
LIN {X 0,Y 441.198,Z 460.526,A -85,B 0,C 180,E1 21026.273,E2 21026.273} C_VEL
LIN {X 0,Y 441.154,Z 460.528,A -85,B 0,C 180,E1 21022.49,E2 21022.49} C_VEL
LIN {X 0,Y 441.172,Z 460.524,A -85,B 0,C 180,E1 21018.737,E2 21018.737} C_VEL
LIN {X 0,Y 441.191,Z 460.534,A -85,B 0,C 180,E1 21014.997,E2 21014.997} C_VEL
LIN {X 0,Y 441.184,Z 460.552,A -85,B 0,C 180,E1 21013.547,E2 21013.547} C_VEL
LIN {X 0,Y 442.509,Z 464.079,A -85,B 0,C 180,E1 21013.029,E2 21013.029} C_VEL
LIN {X 0,Y 449.497,Z 479.741,A -85,B 0,C 180,E1 21010.666,E2 21010.666} C_VEL
LIN {X 0,Y 456.827,Z 498.014,A -85,B 0,C 180,E1 21008.21,E2 21008.21} C_VEL
LIN {X 0,Y 458.02,Z 500.526,A -85,B 0,C 180,E1 21007.969,E2 21007.969} C_VEL
LIN {X 0,Y 462.064,Z 508.348,A -85,B 0,C 180,E1 21007.425,E2 21007.425} C_VEL
LIN {X 0,Y 464.959,Z 525.456,A -85,B 0,C 180,E1 21006.824,E2 21006.824} C_VEL
LIN {X 0,Y 461.18,Z 696.611,A -85,B 0,C 180,E1 21003.951,E2 21003.951} C_VEL
LIN {X 0,Y 460.177,Z 704.301,A -85,B 0,C 180,E1 21003.893,E2 21003.893} C_VEL
LIN {X 0,Y 454.568,Z 724.783,A -85,B 0,C 180,E1 21003.989,E2 21003.989} C_VEL
LIN {X 0,Y 453.812,Z 731.382,A -85,B 0,C 180,E1 21003.93,E2 21003.93} C_VEL
LIN {X 0,Y 452.952,Z 764.176,A -85,B 0,C 180,E1 21003.328,E2 21003.328} C_VEL
LIN {X 0,Y 451.798,Z 785.438,A -85,B 0,C 180,E1 21002.696,E2 21002.696} C_VEL
LIN {X 0,Y 450.391,Z 804.602,A -85,B 0,C 180,E1 21001.894,E2 21001.894} C_VEL
LIN {X 0,Y 448.596,Z 824.097,A -85,B 0,C 180,E1 21000.839,E2 21000.839} C_VEL
LIN {X 0,Y 446.6,Z 842.652,A -85,B 0,C 180,E1 20999.581,E2 20999.581} C_VEL
LIN {X 0,Y 444.513,Z 860.016,A -85,B 0,C 180,E1 20998.147,E2 20998.147} C_VEL
LIN {X 0,Y 442.321,Z 876.878,A -85,B 0,C 180,E1 20996.472,E2 20996.472} C_VEL
LIN {X 0,Y 440.119,Z 892.904,A -85,B 0,C 180,E1 20994.565,E2 20994.565} C_VEL
LIN {X 0,Y 438.032,Z 908.031,A -85,B 0,C 180,E1 20992.407,E2 20992.407} C_VEL
LIN {X 0,Y 436.315,Z 920.73,A -85,B 0,C 180,E1 20990.244,E2 20990.244} C_VEL
LIN {X 0,Y 434.883,Z 932.113,A -85,B 0,C 180,E1 20987.943,E2 20987.943} C_VEL
LIN {X 0,Y 433.7,Z 942.66,A -85,B 0,C 180,E1 20985.374,E2 20985.374} C_VEL
LIN {X 0,Y 432.896,Z 951.213,A -85,B 0,C 180,E1 20982.81,E2 20982.81} C_VEL
LIN {X 0,Y 432.402,Z 958.015,A -85,B 0,C 180,E1 20980.255,E2 20980.255} C_VEL
LIN {X 0,Y 432.116,Z 963.389,A -85,B 0,C 180,E1 20977.578,E2 20977.578} C_VEL
LIN {X 0,Y 431.996,Z 967.053,A -85,B 0,C 180,E1 20974.912,E2 20974.912} C_VEL
LIN {X 0,Y 431.96,Z 969.152,A -85,B 0,C 180,E1 20972.254,E2 20972.254} C_VEL
LIN {X 0,Y 431.948,Z 969.734,A -85,B 0,C 180,E1 20969.601,E2 20969.601} C_VEL
LIN {X 0,Y 431.962,Z 968.8,A -85,B 0,C 180,E1 20966.948,E2 20966.948} C_VEL
LIN {X 0,Y 432.013,Z 966.234,A -85,B 0,C 180,E1 20964.288,E2 20964.288} C_VEL
LIN {X 0,Y 432.18,Z 962.077,A -85,B 0,C 180,E1 20961.618,E2 20961.618} C_VEL
LIN {X 0,Y 432.515,Z 956.236,A -85,B 0,C 180,E1 20958.937,E2 20958.937} C_VEL
LIN {X 0,Y 433.097,Z 949.01,A -85,B 0,C 180,E1 20956.379,E2 20956.379} C_VEL
LIN {X 0,Y 433.998,Z 939.96,A -85,B 0,C 180,E1 20953.813,E2 20953.813} C_VEL
LIN {X 0,Y 435.3,Z 928.8,A -85,B 0,C 180,E1 20951.241,E2 20951.241} C_VEL
LIN {X 0,Y 436.957,Z 915.963,A -85,B 0,C 180,E1 20948.804,E2 20948.804} C_VEL
LIN {X 0,Y 438.815,Z 902.294,A -85,B 0,C 180,E1 20946.642,E2 20946.642} C_VEL
LIN {X 0,Y 440.864,Z 887.466,A -85,B 0,C 180,E1 20944.666,E2 20944.666} C_VEL
LIN {X 0,Y 443.014,Z 871.518,A -85,B 0,C 180,E1 20942.876,E2 20942.876} C_VEL
LIN {X 0,Y 445.293,Z 853.665,A -85,B 0,C 180,E1 20941.207,E2 20941.207} C_VEL
LIN {X 0,Y 447.412,Z 835.539,A -85,B 0,C 180,E1 20939.812,E2 20939.812} C_VEL
LIN {X 0,Y 449.262,Z 817.707,A -85,B 0,C 180,E1 20938.689,E2 20938.689} C_VEL
LIN {X 0,Y 450.943,Z 797.765,A -85,B 0,C 180,E1 20937.699,E2 20937.699} C_VEL
LIN {X 0,Y 452.274,Z 777.758,A -85,B 0,C 180,E1 20936.959,E2 20936.959} C_VEL
LIN {X 0,Y 453.179,Z 757.309,A -85,B 0,C 180,E1 20936.434,E2 20936.434} C_VEL
LIN {X 0,Y 458.245,Z 535.422,A -85,B 0,C 180,E1 20932.639,E2 20932.639} C_VEL
LIN {X 0,Y 451.015,Z 508.688,A -85,B 0,C 180,E1 20931.395,E2 20931.395} C_VEL
LIN {X 0,Y 447.301,Z 501.77,A -85,B 0,C 180,E1 20930.865,E2 20930.865} C_VEL
LIN {X 0,Y 441.893,Z 485.101,A -85,B 0,C 180,E1 20927.951,E2 20927.951} C_VEL
LIN {X 0,Y 437.057,Z 471.586,A -85,B 0,C 180,E1 20925.356,E2 20925.356} C_VEL
LIN {X 0,Y 433.252,Z 461.517,A -85,B 0,C 180,E1 20923.269,E2 20923.269} C_VEL
LIN {X 0,Y 433.247,Z 461.52,A -85,B 0,C 180,E1 20919.566,E2 20919.566} C_VEL
LIN {X 0,Y 433.27,Z 461.643,A -85,B 0,C 180,E1 20918.626,E2 20918.626} C_VEL
LIN {X 0,Y 441.295,Z 482.727,A -85,B 0,C 180,E1 20915.121,E2 20915.121} C_VEL
LIN {X 0,Y 448.072,Z 502.063,A -85,B 0,C 180,E1 20912.129,E2 20912.129} C_VEL
LIN {X 0,Y 449.594,Z 507.484,A -85,B 0,C 180,E1 20911.351,E2 20911.351} C_VEL
LIN {X 0,Y 447.101,Z 541.25,A -85,B 0,C 180,E1 20907.676,E2 20907.676} C_VEL
LIN {X 0,Y 444.622,Z 576.863,A -85,B 0,C 180,E1 20903.878,E2 20903.878} C_VEL
LIN {X 0,Y 442.394,Z 613.757,A -85,B 0,C 180,E1 20900.009,E2 20900.009} C_VEL
LIN {X 0,Y 442.214,Z 619.244,A -85,B 0,C 180,E1 20899.477,E2 20899.477} C_VEL
LIN {X 0,Y 442.885,Z 625.399,A -85,B 0,C 180,E1 20899.296,E2 20899.296} C_VEL
LIN {X 0,Y 439.198,Z 761.678,A -85,B 0,C 180,E1 20896.35,E2 20896.35} C_VEL
LIN {X 0,Y 438.83,Z 778.752,A -85,B 0,C 180,E1 20895.732,E2 20895.732} C_VEL
LIN {X 0,Y 438.285,Z 794.051,A -85,B 0,C 180,E1 20894.939,E2 20894.939} C_VEL
LIN {X 0,Y 437.58,Z 809.315,A -85,B 0,C 180,E1 20893.882,E2 20893.882} C_VEL
LIN {X 0,Y 436.826,Z 822.802,A -85,B 0,C 180,E1 20892.694,E2 20892.694} C_VEL
LIN {X 0,Y 435.959,Z 836.483,A -85,B 0,C 180,E1 20891.175,E2 20891.175} C_VEL
LIN {X 0,Y 435.234,Z 847.501,A -85,B 0,C 180,E1 20889.654,E2 20889.654} C_VEL
LIN {X 0,Y 434.525,Z 858.259,A -85,B 0,C 180,E1 20887.803,E2 20887.803} C_VEL
LIN {X 0,Y 434,Z 866.767,A -85,B 0,C 180,E1 20885.951,E2 20885.951} C_VEL
LIN {X 0,Y 433.594,Z 874.252,A -85,B 0,C 180,E1 20883.835,E2 20883.835} C_VEL
LIN {X 0,Y 433.356,Z 879.367,A -85,B 0,C 180,E1 20881.851,E2 20881.851} C_VEL
LIN {X 0,Y 433.255,Z 883.219,A -85,B 0,C 180,E1 20879.604,E2 20879.604} C_VEL
LIN {X 0,Y 433.259,Z 885.04,A -85,B 0,C 180,E1 20877.487,E2 20877.487} C_VEL
LIN {X 0,Y 433.391,Z 885.155,A -85,B 0,C 180,E1 20875.236,E2 20875.236} C_VEL
LIN {X 0,Y 433.621,Z 883.457,A -85,B 0,C 180,E1 20873.114,E2 20873.114} C_VEL
LIN {X 0,Y 434.02,Z 880.061,A -85,B 0,C 180,E1 20870.988,E2 20870.988} C_VEL
LIN {X 0,Y 434.587,Z 874.678,A -85,B 0,C 180,E1 20868.857,E2 20868.857} C_VEL
LIN {X 0,Y 435.322,Z 867.742,A -85,B 0,C 180,E1 20866.857,E2 20866.857} C_VEL
LIN {X 0,Y 436.269,Z 858.551,A -85,B 0,C 180,E1 20864.855,E2 20864.855} C_VEL
LIN {X 0,Y 437.191,Z 849.121,A -85,B 0,C 180,E1 20863.252,E2 20863.252} C_VEL
LIN {X 0,Y 438.292,Z 837.203,A -85,B 0,C 180,E1 20861.626,E2 20861.626} C_VEL
LIN {X 0,Y 439.289,Z 824.338,A -85,B 0,C 180,E1 20860.245,E2 20860.245} C_VEL
LIN {X 0,Y 440.149,Z 810.92,A -85,B 0,C 180,E1 20859.106,E2 20859.106} C_VEL
LIN {X 0,Y 440.874,Z 795.358,A -85,B 0,C 180,E1 20858.095,E2 20858.095} C_VEL
LIN {X 0,Y 441.288,Z 779.812,A -85,B 0,C 180,E1 20857.372,E2 20857.372} C_VEL
LIN {X 0,Y 441.994,Z 750.093,A -85,B 0,C 180,E1 20856.446,E2 20856.446} C_VEL
LIN {X 0,Y 448.085,Z 665.142,A -85,B 0,C 180,E1 20853.905,E2 20853.905} C_VEL
LIN {X 0,Y 449.689,Z 647.55,A -85,B 0,C 180,E1 20853.359,E2 20853.359} C_VEL
LIN {X 0,Y 455.27,Z 635.371,A -85,B 0,C 180,E1 20852.323,E2 20852.323} C_VEL
LIN {X 0,Y 461.312,Z 610.442,A -85,B 0,C 180,E1 20848.946,E2 20848.946} C_VEL
LIN {X 0,Y 468.427,Z 589.771,A -85,B 0,C 180,E1 20845.914,E2 20845.914} C_VEL
LIN {X 0,Y 476.252,Z 573.6,A -85,B 0,C 180,E1 20843.321,E2 20843.321} C_VEL
LIN {X 0,Y 481.521,Z 565.337,A -85,B 0,C 180,E1 20841.862,E2 20841.862} C_VEL
LIN {X 0,Y 473.248,Z 577.322,A -85,B 0,C 180,E1 20840.269,E2 20840.269} C_VEL
LIN {X 0,Y 466.986,Z 589.69,A -85,B 0,C 180,E1 20838.631,E2 20838.631} C_VEL
LIN {X 0,Y 462.618,Z 603.1,A -85,B 0,C 180,E1 20836.84,E2 20836.84} C_VEL
LIN {X 0,Y 460.795,Z 615.939,A -85,B 0,C 180,E1 20835.111,E2 20835.111} C_VEL
LIN {X 0,Y 461.257,Z 628.814,A -85,B 0,C 180,E1 20833.343,E2 20833.343} C_VEL
LIN {X 0,Y 464.067,Z 641.375,A -85,B 0,C 180,E1 20831.615,E2 20831.615} C_VEL
LIN {X 0,Y 468.824,Z 652.718,A -85,B 0,C 180,E1 20830.037,E2 20830.037} C_VEL
LIN {X 0,Y 476.087,Z 664.21,A -85,B 0,C 180,E1 20828.431,E2 20828.431} C_VEL
LIN {X 0,Y 485.419,Z 674.789,A -85,B 0,C 180,E1 20826.947,E2 20826.947} C_VEL
LIN {X 0,Y 488.697,Z 677.964,A -85,B 0,C 180,E1 20826.508,E2 20826.508} C_VEL
LIN {X 0,Y 476.13,Z 697.184,A -85,B 0,C 180,E1 20825.867,E2 20825.867} C_VEL
LIN {X 0,Y 466.884,Z 714.001,A -85,B 0,C 180,E1 20825.176,E2 20825.176} C_VEL
LIN {X 0,Y 459.995,Z 729.62,A -85,B 0,C 180,E1 20824.413,E2 20824.413} C_VEL
LIN {X 0,Y 457.074,Z 736.878,A -85,B 0,C 180,E1 20824.071,E2 20824.071} C_VEL
LIN {X 0,Y 454.288,Z 755.577,A -85,B 0,C 180,E1 20823.959,E2 20823.959} C_VEL
LIN {X 0,Y 452.464,Z 774.567,A -85,B 0,C 180,E1 20823.76,E2 20823.76} C_VEL
LIN {X 0,Y 451.563,Z 805.024,A -85,B 0,C 180,E1 20823.199,E2 20823.199} C_VEL
LIN {X 0,Y 450.352,Z 825.615,A -85,B 0,C 180,E1 20822.603,E2 20822.603} C_VEL
LIN {X 0,Y 448.716,Z 846.143,A -85,B 0,C 180,E1 20821.765,E2 20821.765} C_VEL
LIN {X 0,Y 446.935,Z 865.08,A -85,B 0,C 180,E1 20820.744,E2 20820.744} C_VEL
LIN {X 0,Y 444.915,Z 883.859,A -85,B 0,C 180,E1 20819.483,E2 20819.483} C_VEL
LIN {X 0,Y 442.764,Z 901.996,A -85,B 0,C 180,E1 20817.998,E2 20817.998} C_VEL
LIN {X 0,Y 440.718,Z 918.784,A -85,B 0,C 180,E1 20816.346,E2 20816.346} C_VEL
LIN {X 0,Y 438.749,Z 934.564,A -85,B 0,C 180,E1 20814.505,E2 20814.505} C_VEL
LIN {X 0,Y 436.892,Z 949.789,A -85,B 0,C 180,E1 20812.395,E2 20812.395} C_VEL
LIN {X 0,Y 435.252,Z 964.147,A -85,B 0,C 180,E1 20810.017,E2 20810.017} C_VEL
LIN {X 0,Y 433.99,Z 976.462,A -85,B 0,C 180,E1 20807.567,E2 20807.567} C_VEL
LIN {X 0,Y 433.124,Z 986.663,A -85,B 0,C 180,E1 20805.122,E2 20805.122} C_VEL
LIN {X 0,Y 432.552,Z 995.459,A -85,B 0,C 180,E1 20802.55,E2 20802.55} C_VEL
LIN {X 0,Y 432.24,Z 1002.755,A -85,B 0,C 180,E1 20799.857,E2 20799.857} C_VEL
LIN {X 0,Y 432.103,Z 1007.987,A -85,B 0,C 180,E1 20797.312,E2 20797.312} C_VEL
LIN {X 0,Y 432.101,Z 1011.583,A -85,B 0,C 180,E1 20794.779,E2 20794.779} C_VEL
LIN {X 0,Y 432.121,Z 1013.636,A -85,B 0,C 180,E1 20792.255,E2 20792.255} C_VEL
LIN {X 0,Y 432.126,Z 1014.227,A -85,B 0,C 180,E1 20789.603,E2 20789.603} C_VEL
LIN {X 0,Y 432.107,Z 1013.283,A -85,B 0,C 180,E1 20787.083,E2 20787.083} C_VEL
LIN {X 0,Y 432.084,Z 1010.762,A -85,B 0,C 180,E1 20784.557,E2 20784.557} C_VEL
LIN {X 0,Y 432.13,Z 1006.49,A -85,B 0,C 180,E1 20781.887,E2 20781.887} C_VEL
LIN {X 0,Y 432.29,Z 1000.804,A -85,B 0,C 180,E1 20779.338,E2 20779.338} C_VEL
LIN {X 0,Y 432.656,Z 993.391,A -85,B 0,C 180,E1 20776.775,E2 20776.775} C_VEL
LIN {X 0,Y 433.31,Z 984.039,A -85,B 0,C 180,E1 20774.201,E2 20774.201} C_VEL
LIN {X 0,Y 434.254,Z 973.23,A -85,B 0,C 180,E1 20771.752,E2 20771.752} C_VEL
LIN {X 0,Y 435.538,Z 961.022,A -85,B 0,C 180,E1 20769.438,E2 20769.438} C_VEL
LIN {X 0,Y 437.185,Z 946.819,A -85,B 0,C 180,E1 20767.172,E2 20767.172} C_VEL
LIN {X 0,Y 439.041,Z 931.724,A -85,B 0,C 180,E1 20765.142,E2 20765.142} C_VEL
LIN {X 0,Y 441.054,Z 915.789,A -85,B 0,C 180,E1 20763.33,E2 20763.33} C_VEL
LIN {X 0,Y 443.241,Z 897.707,A -85,B 0,C 180,E1 20761.613,E2 20761.613} C_VEL
LIN {X 0,Y 445.368,Z 879.319,A -85,B 0,C 180,E1 20760.181,E2 20760.181} C_VEL
LIN {X 0,Y 447.307,Z 860.525,A -85,B 0,C 180,E1 20758.988,E2 20758.988} C_VEL
LIN {X 0,Y 449.083,Z 840.948,A -85,B 0,C 180,E1 20758.003,E2 20758.003} C_VEL
LIN {X 0,Y 450.617,Z 820.187,A -85,B 0,C 180,E1 20757.217,E2 20757.217} C_VEL
LIN {X 0,Y 451.737,Z 799.529,A -85,B 0,C 180,E1 20756.677,E2 20756.677} C_VEL
LIN {X 0,Y 452.768,Z 768.12,A -85,B 0,C 180,E1 20756.149,E2 20756.149} C_VEL
LIN {X 0,Y 454.083,Z 755.594,A -85,B 0,C 180,E1 20755.994,E2 20755.994} C_VEL
LIN {X 0,Y 459.862,Z 740.636,A -85,B 0,C 180,E1 20755.18,E2 20755.18} C_VEL
LIN {X 0,Y 469.647,Z 718.507,A -85,B 0,C 180,E1 20754.09,E2 20754.09} C_VEL
LIN {X 0,Y 478.914,Z 701.634,A -85,B 0,C 180,E1 20753.413,E2 20753.413} C_VEL
LIN {X 0,Y 491.275,Z 682.584,A -85,B 0,C 180,E1 20752.81,E2 20752.81} C_VEL
LIN {X 0,Y 491.907,Z 681.667,A -85,B 0,C 180,E1 20752.786,E2 20752.786} C_VEL
LIN {X 0,Y 481.828,Z 670.903,A -85,B 0,C 180,E1 20751.194,E2 20751.194} C_VEL
LIN {X 0,Y 473.866,Z 659.12,A -85,B 0,C 180,E1 20749.615,E2 20749.615} C_VEL
LIN {X 0,Y 467.799,Z 646.469,A -85,B 0,C 180,E1 20748.056,E2 20748.056} C_VEL
LIN {X 0,Y 463.263,Z 631.765,A -85,B 0,C 180,E1 20746.394,E2 20746.394} C_VEL
LIN {X 0,Y 460.534,Z 615.527,A -85,B 0,C 180,E1 20744.703,E2 20744.703} C_VEL
LIN {X 0,Y 459.718,Z 597.693,A -85,B 0,C 180,E1 20742.996,E2 20742.996} C_VEL
LIN {X 0,Y 460.974,Z 574.804,A -85,B 0,C 180,E1 20740.992,E2 20740.992} C_VEL
LIN {X 0,Y 465.073,Z 536.831,A -85,B 0,C 180,E1 20737.786,E2 20737.786} C_VEL
LIN {X 0,Y 466.009,Z 528.569,A -85,B 0,C 180,E1 20737.078,E2 20737.078} C_VEL
LIN {X 0,Y 456.434,Z 508.335,A -85,B 0,C 180,E1 20733.808,E2 20733.808} C_VEL
LIN {X 0,Y 447.896,Z 490.977,A -85,B 0,C 180,E1 20730.744,E2 20730.744} C_VEL
LIN {X 0,Y 441.591,Z 478.608,A -85,B 0,C 180,E1 20728.391,E2 20728.391} C_VEL
LIN {X 0,Y 437.107,Z 469.84,A -85,B 0,C 180,E1 20726.637,E2 20726.637} C_VEL
LIN {X 0,Y 435.316,Z 465.95,A -85,B 0,C 180,E1 20725.874,E2 20725.874} C_VEL
LIN {X 0,Y 433.628,Z 463.172,A -85,B 0,C 180,E1 20725.25,E2 20725.25} C_VEL
LIN {X 0,Y 433.247,Z 461.519,A -85,B 0,C 180,E1 20724.942,E2 20724.942} C_VEL
LIN {X 0,Y 433.241,Z 461.52,A -85,B 0,C 180,E1 20721.194,E2 20721.194} C_VEL
LIN {X 0,Y 433.246,Z 461.52,A -85,B 0,C 180,E1 20717.32,E2 20717.32} C_VEL
LIN {X 0,Y 433.251,Z 461.521,A -85,B 0,C 180,E1 20713.615,E2 20713.615} C_VEL
LIN {X 0,Y 433.251,Z 461.52,A -85,B 0,C 180,E1 20709.699,E2 20709.699} C_VEL
LIN {X 0,Y 433.237,Z 461.521,A -85,B 0,C 180,E1 20705.911,E2 20705.911} C_VEL
LIN {X 0,Y 433.216,Z 461.523,A -85,B 0,C 180,E1 20701.984,E2 20701.984} C_VEL
LIN {X 0,Y 433.256,Z 461.516,A -85,B 0,C 180,E1 20698.281,E2 20698.281} C_VEL
LIN {X 0,Y 433.231,Z 461.521,A -85,B 0,C 180,E1 20694.57,E2 20694.57} C_VEL
LIN {X 0,Y 433.257,Z 461.511,A -85,B 0,C 180,E1 20690.837,E2 20690.837} C_VEL
LIN {X 0,Y 433.213,Z 461.507,A -85,B 0,C 180,E1 20687.199,E2 20687.199} C_VEL
LIN {X 0,Y 433.241,Z 461.517,A -85,B 0,C 180,E1 20683.509,E2 20683.509} C_VEL
LIN {X 0,Y 433.242,Z 461.522,A -85,B 0,C 180,E1 20679.746,E2 20679.746} C_VEL
LIN {X 0,Y 433.241,Z 461.519,A -85,B 0,C 180,E1 20675.89,E2 20675.89} C_VEL
LIN {X 0,Y 433.261,Z 461.511,A -85,B 0,C 180,E1 20672.064,E2 20672.064} C_VEL
LIN {X 0,Y 433.252,Z 461.511,A -85,B 0,C 180,E1 20668.252,E2 20668.252} C_VEL
LIN {X 0,Y 433.245,Z 461.515,A -85,B 0,C 180,E1 20664.553,E2 20664.553} C_VEL
LIN {X 0,Y 433.211,Z 461.524,A -85,B 0,C 180,E1 20660.602,E2 20660.602} C_VEL
LIN {X 0,Y 433.255,Z 461.514,A -85,B 0,C 180,E1 20656.823,E2 20656.823} C_VEL
LIN {X 0,Y 433.239,Z 461.665,A -85,B 0,C 180,E1 20654.419,E2 20654.419} C_VEL
LIN {X 0,Y 434.489,Z 464.941,A -85,B 0,C 180,E1 20653.922,E2 20653.922} C_VEL
LIN {X 0,Y 440.497,Z 478.033,A -85,B 0,C 180,E1 20651.861,E2 20651.861} C_VEL
LIN {X 0,Y 447.537,Z 494.818,A -85,B 0,C 180,E1 20649.475,E2 20649.475} C_VEL
LIN {X 0,Y 449.751,Z 500.155,A -85,B 0,C 180,E1 20648.811,E2 20648.811} C_VEL
LIN {X 0,Y 456.078,Z 511.907,A -85,B 0,C 180,E1 20647.937,E2 20647.937} C_VEL
LIN {X 0,Y 458.55,Z 527.013,A -85,B 0,C 180,E1 20647.401,E2 20647.401} C_VEL
LIN {X 0,Y 453.812,Z 731.382,A -85,B 0,C 180,E1 20643.93,E2 20643.93} C_VEL
LIN {X 0,Y 452.848,Z 739.077,A -85,B 0,C 180,E1 20643.874,E2 20643.874} C_VEL
LIN {X 0,Y 447.151,Z 759.531,A -85,B 0,C 180,E1 20643.955,E2 20643.955} C_VEL
LIN {X 0,Y 446.206,Z 766.063,A -85,B 0,C 180,E1 20643.851,E2 20643.851} C_VEL
LIN {X 0,Y 445.014,Z 786.968,A -85,B 0,C 180,E1 20643.211,E2 20643.211} C_VEL
LIN {X 0,Y 443.439,Z 807.12,A -85,B 0,C 180,E1 20642.339,E2 20642.339} C_VEL
LIN {X 0,Y 441.497,Z 826.677,A -85,B 0,C 180,E1 20641.239,E2 20641.239} C_VEL
LIN {X 0,Y 439.407,Z 844.8,A -85,B 0,C 180,E1 20639.964,E2 20639.964} C_VEL
LIN {X 0,Y 437.072,Z 862.886,A -85,B 0,C 180,E1 20638.412,E2 20638.412} C_VEL
LIN {X 0,Y 434.707,Z 879.889,A -85,B 0,C 180,E1 20636.648,E2 20636.648} C_VEL
LIN {X 0,Y 432.454,Z 895.303,A -85,B 0,C 180,E1 20634.738,E2 20634.738} C_VEL
LIN {X 0,Y 430.413,Z 909.309,A -85,B 0,C 180,E1 20632.682,E2 20632.682} C_VEL
LIN {X 0,Y 428.507,Z 922.64,A -85,B 0,C 180,E1 20630.344,E2 20630.344} C_VEL
LIN {X 0,Y 426.935,Z 934.378,A -85,B 0,C 180,E1 20627.865,E2 20627.865} C_VEL
LIN {X 0,Y 425.775,Z 944.072,A -85,B 0,C 180,E1 20625.388,E2 20625.388} C_VEL
LIN {X 0,Y 424.935,Z 952.411,A -85,B 0,C 180,E1 20622.778,E2 20622.778} C_VEL
LIN {X 0,Y 424.4,Z 959.374,A -85,B 0,C 180,E1 20620.008,E2 20620.008} C_VEL
LIN {X 0,Y 424.119,Z 964.442,A -85,B 0,C 180,E1 20617.313,E2 20617.313} C_VEL
LIN {X 0,Y 424.009,Z 967.927,A -85,B 0,C 180,E1 20614.598,E2 20614.598} C_VEL
LIN {X 0,Y 423.968,Z 969.761,A -85,B 0,C 180,E1 20611.891,E2 20611.891} C_VEL
LIN {X 0,Y 423.962,Z 970.079,A -85,B 0,C 180,E1 20609.189,E2 20609.189} C_VEL
LIN {X 0,Y 423.976,Z 968.89,A -85,B 0,C 180,E1 20606.484,E2 20606.484} C_VEL
LIN {X 0,Y 424.068,Z 966.165,A -85,B 0,C 180,E1 20603.773,E2 20603.773} C_VEL
LIN {X 0,Y 424.286,Z 961.475,A -85,B 0,C 180,E1 20600.897,E2 20600.897} C_VEL
LIN {X 0,Y 424.696,Z 955.281,A -85,B 0,C 180,E1 20598.18,E2 20598.18} C_VEL
LIN {X 0,Y 425.412,Z 947.552,A -85,B 0,C 180,E1 20595.544,E2 20595.544} C_VEL
LIN {X 0,Y 426.462,Z 938.145,A -85,B 0,C 180,E1 20592.958,E2 20592.958} C_VEL
LIN {X 0,Y 427.875,Z 927.173,A -85,B 0,C 180,E1 20590.478,E2 20590.478} C_VEL
LIN {X 0,Y 429.617,Z 914.752,A -85,B 0,C 180,E1 20588.137,E2 20588.137} C_VEL
LIN {X 0,Y 431.655,Z 900.849,A -85,B 0,C 180,E1 20585.94,E2 20585.94} C_VEL
LIN {X 0,Y 433.936,Z 885.336,A -85,B 0,C 180,E1 20583.889,E2 20583.889} C_VEL
LIN {X 0,Y 436.314,Z 868.66,A -85,B 0,C 180,E1 20582.054,E2 20582.054} C_VEL
LIN {X 0,Y 438.612,Z 851.172,A -85,B 0,C 180,E1 20580.453,E2 20580.453} C_VEL
LIN {X 0,Y 440.813,Z 832.989,A -85,B 0,C 180,E1 20579.085,E2 20579.085} C_VEL
LIN {X 0,Y 442.754,Z 814.341,A -85,B 0,C 180,E1 20577.947,E2 20577.947} C_VEL
LIN {X 0,Y 444.462,Z 794.574,A -85,B 0,C 180,E1 20577.001,E2 20577.001} C_VEL
LIN {X 0,Y 445.787,Z 774.734,A -85,B 0,C 180,E1 20576.292,E2 20576.292} C_VEL
LIN {X 0,Y 446.701,Z 753.352,A -85,B 0,C 180,E1 20575.779,E2 20575.779} C_VEL
LIN {X 0,Y 451.883,Z 537.285,A -85,B 0,C 180,E1 20572.053,E2 20572.053} C_VEL
LIN {X 0,Y 445.238,Z 512.626,A -85,B 0,C 180,E1 20570.875,E2 20570.875} C_VEL
LIN {X 0,Y 439.349,Z 501.88,A -85,B 0,C 180,E1 20569.978,E2 20569.978} C_VEL
LIN {X 0,Y 434.035,Z 485.842,A -85,B 0,C 180,E1 20567.101,E2 20567.101} C_VEL
LIN {X 0,Y 429.279,Z 472.744,A -85,B 0,C 180,E1 20564.514,E2 20564.514} C_VEL
LIN {X 0,Y 425.315,Z 462.502,A -85,B 0,C 180,E1 20562.339,E2 20562.339} C_VEL
LIN {X 0,Y 425.327,Z 462.62,A -85,B 0,C 180,E1 20559.421,E2 20559.421} C_VEL
LIN {X 0,Y 433.069,Z 482.738,A -85,B 0,C 180,E1 20555.978,E2 20555.978} C_VEL
LIN {X 0,Y 439.966,Z 502.147,A -85,B 0,C 180,E1 20552.898,E2 20552.898} C_VEL
LIN {X 0,Y 442.506,Z 510.181,A -85,B 0,C 180,E1 20551.692,E2 20551.692} C_VEL
LIN {X 0,Y 439.852,Z 544.545,A -85,B 0,C 180,E1 20547.923,E2 20547.923} C_VEL
LIN {X 0,Y 437.267,Z 580.08,A -85,B 0,C 180,E1 20544.09,E2 20544.09} C_VEL
LIN {X 0,Y 434.951,Z 616.437,A -85,B 0,C 180,E1 20540.241,E2 20540.241} C_VEL
LIN {X 0,Y 434.843,Z 620.181,A -85,B 0,C 180,E1 20539.884,E2 20539.884} C_VEL
LIN {X 0,Y 435.521,Z 626.446,A -85,B 0,C 180,E1 20539.693,E2 20539.693} C_VEL
LIN {X 0,Y 431.599,Z 762.551,A -85,B 0,C 180,E1 20536.664,E2 20536.664} C_VEL
LIN {X 0,Y 431.213,Z 779.477,A -85,B 0,C 180,E1 20536.04,E2 20536.04} C_VEL
LIN {X 0,Y 430.626,Z 795.191,A -85,B 0,C 180,E1 20535.211,E2 20535.211} C_VEL
LIN {X 0,Y 429.846,Z 811.223,A -85,B 0,C 180,E1 20534.072,E2 20534.072} C_VEL
LIN {X 0,Y 429.008,Z 825.193,A -85,B 0,C 180,E1 20532.792,E2 20532.792} C_VEL
LIN {X 0,Y 428.152,Z 838.128,A -85,B 0,C 180,E1 20531.313,E2 20531.313} C_VEL
LIN {X 0,Y 427.365,Z 849.462,A -85,B 0,C 180,E1 20529.698,E2 20529.698} C_VEL
LIN {X 0,Y 426.639,Z 860.107,A -85,B 0,C 180,E1 20527.812,E2 20527.812} C_VEL
LIN {X 0,Y 426.099,Z 868.469,A -85,B 0,C 180,E1 20525.926,E2 20525.926} C_VEL
LIN {X 0,Y 425.703,Z 875.46,A -85,B 0,C 180,E1 20523.906,E2 20523.906} C_VEL
LIN {X 0,Y 425.456,Z 880.608,A -85,B 0,C 180,E1 20521.886,E2 20521.886} C_VEL
LIN {X 0,Y 425.353,Z 884.5,A -85,B 0,C 180,E1 20519.596,E2 20519.596} C_VEL
LIN {X 0,Y 425.366,Z 886.35,A -85,B 0,C 180,E1 20517.44,E2 20517.44} C_VEL
LIN {X 0,Y 425.516,Z 886.502,A -85,B 0,C 180,E1 20515.148,E2 20515.148} C_VEL
LIN {X 0,Y 425.778,Z 884.828,A -85,B 0,C 180,E1 20512.986,E2 20512.986} C_VEL
LIN {X 0,Y 426.219,Z 881.466,A -85,B 0,C 180,E1 20510.821,E2 20510.821} C_VEL
LIN {X 0,Y 426.851,Z 876.132,A -85,B 0,C 180,E1 20508.653,E2 20508.653} C_VEL
LIN {X 0,Y 427.598,Z 869.77,A -85,B 0,C 180,E1 20506.753,E2 20506.753} C_VEL
LIN {X 0,Y 428.527,Z 861.406,A -85,B 0,C 180,E1 20504.852,E2 20504.852} C_VEL
LIN {X 0,Y 429.604,Z 851.61,A -85,B 0,C 180,E1 20503.087,E2 20503.087} C_VEL
LIN {X 0,Y 430.805,Z 839.622,A -85,B 0,C 180,E1 20501.39,E2 20501.39} C_VEL
LIN {X 0,Y 431.82,Z 827.831,A -85,B 0,C 180,E1 20500.066,E2 20500.066} C_VEL
LIN {X 0,Y 432.786,Z 814.65,A -85,B 0,C 180,E1 20498.875,E2 20498.875} C_VEL
LIN {X 0,Y 433.517,Z 801.007,A -85,B 0,C 180,E1 20497.918,E2 20497.918} C_VEL
LIN {X 0,Y 434.101,Z 785.094,A -85,B 0,C 180,E1 20497.083,E2 20497.083} C_VEL
LIN {X 0,Y 434.507,Z 763.868,A -85,B 0,C 180,E1 20496.338,E2 20496.338} C_VEL
LIN {X 0,Y 437.671,Z 715.212,A -85,B 0,C 180,E1 20494.814,E2 20494.814} C_VEL
LIN {X 0,Y 443.464,Z 650.652,A -85,B 0,C 180,E1 20492.762,E2 20492.762} C_VEL
LIN {X 0,Y 449.565,Z 637.691,A -85,B 0,C 180,E1 20491.652,E2 20491.652} C_VEL
LIN {X 0,Y 456.132,Z 613.424,A -85,B 0,C 180,E1 20488.269,E2 20488.269} C_VEL
LIN {X 0,Y 463.67,Z 593.818,A -85,B 0,C 180,E1 20485.299,E2 20485.299} C_VEL
LIN {X 0,Y 471.661,Z 578.916,A -85,B 0,C 180,E1 20482.832,E2 20482.832} C_VEL
LIN {X 0,Y 474.815,Z 574.22,A -85,B 0,C 180,E1 20481.959,E2 20481.959} C_VEL
LIN {X 0,Y 466.512,Z 586.328,A -85,B 0,C 180,E1 20480.304,E2 20480.304} C_VEL
LIN {X 0,Y 460.441,Z 598.541,A -85,B 0,C 180,E1 20478.614,E2 20478.614} C_VEL
LIN {X 0,Y 456.459,Z 611.244,A -85,B 0,C 180,E1 20476.839,E2 20476.839} C_VEL
LIN {X 0,Y 454.9,Z 623.843,A -85,B 0,C 180,E1 20475.053,E2 20475.053} C_VEL
LIN {X 0,Y 455.703,Z 636.739,A -85,B 0,C 180,E1 20473.202,E2 20473.202} C_VEL
LIN {X 0,Y 458.844,Z 648.943,A -85,B 0,C 180,E1 20471.444,E2 20471.444} C_VEL
LIN {X 0,Y 464.272,Z 660.643,A -85,B 0,C 180,E1 20469.751,E2 20469.751} C_VEL
LIN {X 0,Y 471.775,Z 671.655,A -85,B 0,C 180,E1 20468.161,E2 20468.161} C_VEL
LIN {X 0,Y 479.498,Z 680.211,A -85,B 0,C 180,E1 20466.928,E2 20466.928} C_VEL
LIN {X 0,Y 467.383,Z 699.458,A -85,B 0,C 180,E1 20466.265,E2 20466.265} C_VEL
LIN {X 0,Y 458.451,Z 716.458,A -85,B 0,C 180,E1 20465.537,E2 20465.537} C_VEL
LIN {X 0,Y 450.824,Z 734.578,A -85,B 0,C 180,E1 20464.649,E2 20464.649} C_VEL
LIN {X 0,Y 447.868,Z 753.691,A -85,B 0,C 180,E1 20464.546,E2 20464.546} C_VEL
LIN {X 0,Y 445.848,Z 773.954,A -85,B 0,C 180,E1 20464.337,E2 20464.337} C_VEL
LIN {X 0,Y 444.884,Z 804.423,A -85,B 0,C 180,E1 20463.772,E2 20463.772} C_VEL
LIN {X 0,Y 443.595,Z 825.161,A -85,B 0,C 180,E1 20463.168,E2 20463.168} C_VEL
LIN {X 0,Y 441.922,Z 845.042,A -85,B 0,C 180,E1 20462.351,E2 20462.351} C_VEL
LIN {X 0,Y 440,Z 864.378,A -85,B 0,C 180,E1 20461.304,E2 20461.304} C_VEL
LIN {X 0,Y 437.972,Z 882.351,A -85,B 0,C 180,E1 20460.091,E2 20460.091} C_VEL
LIN {X 0,Y 435.664,Z 900.675,A -85,B 0,C 180,E1 20458.589,E2 20458.589} C_VEL
LIN {X 0,Y 433.553,Z 917.077,A -85,B 0,C 180,E1 20456.972,E2 20456.972} C_VEL
LIN {X 0,Y 431.407,Z 933.098,A -85,B 0,C 180,E1 20455.097,E2 20455.097} C_VEL
LIN {X 0,Y 429.456,Z 947.944,A -85,B 0,C 180,E1 20453.026,E2 20453.026} C_VEL
LIN {X 0,Y 427.757,Z 961.579,A -85,B 0,C 180,E1 20450.776,E2 20450.776} C_VEL
LIN {X 0,Y 426.399,Z 973.454,A -85,B 0,C 180,E1 20448.456,E2 20448.456} C_VEL
LIN {X 0,Y 425.411,Z 984.144,A -85,B 0,C 180,E1 20445.962,E2 20445.962} C_VEL
LIN {X 0,Y 424.705,Z 993.384,A -85,B 0,C 180,E1 20443.34,E2 20443.34} C_VEL
LIN {X 0,Y 424.296,Z 1001.09,A -85,B 0,C 180,E1 20440.592,E2 20440.592} C_VEL
LIN {X 0,Y 424.143,Z 1006.856,A -85,B 0,C 180,E1 20437.859,E2 20437.859} C_VEL
LIN {X 0,Y 424.094,Z 1010.678,A -85,B 0,C 180,E1 20435.276,E2 20435.276} C_VEL
LIN {X 0,Y 424.124,Z 1013.084,A -85,B 0,C 180,E1 20432.568,E2 20432.568} C_VEL
LIN {X 0,Y 424.151,Z 1013.878,A -85,B 0,C 180,E1 20430.001,E2 20430.001} C_VEL
LIN {X 0,Y 424.12,Z 1013.013,A -85,B 0,C 180,E1 20427.298,E2 20427.298} C_VEL
LIN {X 0,Y 424.09,Z 1010.513,A -85,B 0,C 180,E1 20424.589,E2 20424.589} C_VEL
LIN {X 0,Y 424.132,Z 1006.337,A -85,B 0,C 180,E1 20421.869,E2 20421.869} C_VEL
LIN {X 0,Y 424.297,Z 1000.75,A -85,B 0,C 180,E1 20419.272,E2 20419.272} C_VEL
LIN {X 0,Y 424.704,Z 992.975,A -85,B 0,C 180,E1 20416.523,E2 20416.523} C_VEL
LIN {X 0,Y 425.423,Z 983.623,A -85,B 0,C 180,E1 20413.9,E2 20413.9} C_VEL
LIN {X 0,Y 426.444,Z 972.813,A -85,B 0,C 180,E1 20411.406,E2 20411.406} C_VEL
LIN {X 0,Y 427.825,Z 960.604,A -85,B 0,C 180,E1 20409.05,E2 20409.05} C_VEL
LIN {X 0,Y 429.523,Z 947.006,A -85,B 0,C 180,E1 20406.834,E2 20406.834} C_VEL
LIN {X 0,Y 431.497,Z 931.973,A -85,B 0,C 180,E1 20404.764,E2 20404.764} C_VEL
LIN {X 0,Y 433.737,Z 915.38,A -85,B 0,C 180,E1 20402.844,E2 20402.844} C_VEL
LIN {X 0,Y 435.997,Z 897.777,A -85,B 0,C 180,E1 20401.144,E2 20401.144} C_VEL
LIN {X 0,Y 438.314,Z 878.922,A -85,B 0,C 180,E1 20399.651,E2 20399.651} C_VEL
LIN {X 0,Y 440.373,Z 860.137,A -85,B 0,C 180,E1 20398.444,E2 20398.444} C_VEL
LIN {X 0,Y 442.252,Z 840.574,A -85,B 0,C 180,E1 20397.448,E2 20397.448} C_VEL
LIN {X 0,Y 443.861,Z 819.966,A -85,B 0,C 180,E1 20396.658,E2 20396.658} C_VEL
LIN {X 0,Y 445.046,Z 799.335,A -85,B 0,C 180,E1 20396.112,E2 20396.112} C_VEL
LIN {X 0,Y 446.118,Z 768.233,A -85,B 0,C 180,E1 20395.581,E2 20395.581} C_VEL
LIN {X 0,Y 447.533,Z 753.783,A -85,B 0,C 180,E1 20395.426,E2 20395.426} C_VEL
LIN {X 0,Y 453.742,Z 738.285,A -85,B 0,C 180,E1 20394.582,E2 20394.582} C_VEL
LIN {X 0,Y 462.901,Z 717.721,A -85,B 0,C 180,E1 20393.56,E2 20393.56} C_VEL
LIN {X 0,Y 472.594,Z 700.172,A -85,B 0,C 180,E1 20392.842,E2 20392.842} C_VEL
LIN {X 0,Y 482.822,Z 684.005,A -85,B 0,C 180,E1 20392.309,E2 20392.309} C_VEL
LIN {X 0,Y 473.683,Z 673.403,A -85,B 0,C 180,E1 20390.775,E2 20390.775} C_VEL
LIN {X 0,Y 465.725,Z 660.654,A -85,B 0,C 180,E1 20389.087,E2 20389.087} C_VEL
LIN {X 0,Y 459.982,Z 647.382,A -85,B 0,C 180,E1 20387.466,E2 20387.466} C_VEL
LIN {X 0,Y 455.876,Z 632.395,A -85,B 0,C 180,E1 20385.777,E2 20385.777} C_VEL
LIN {X 0,Y 453.463,Z 615.211,A -85,B 0,C 180,E1 20383.992,E2 20383.992} C_VEL
LIN {X 0,Y 453.089,Z 595.618,A -85,B 0,C 180,E1 20382.133,E2 20382.133} C_VEL
LIN {X 0,Y 455.149,Z 569.998,A -85,B 0,C 180,E1 20379.9,E2 20379.9} C_VEL
LIN {X 0,Y 459.113,Z 535.475,A -85,B 0,C 180,E1 20376.942,E2 20376.942} C_VEL
LIN {X 0,Y 459.476,Z 532.416,A -85,B 0,C 180,E1 20376.679,E2 20376.679} C_VEL
LIN {X 0,Y 450.102,Z 512.589,A -85,B 0,C 180,E1 20373.429,E2 20373.429} C_VEL
LIN {X 0,Y 440.98,Z 493.766,A -85,B 0,C 180,E1 20370.072,E2 20370.072} C_VEL
LIN {X 0,Y 433.4,Z 479.073,A -85,B 0,C 180,E1 20367.18,E2 20367.18} C_VEL
LIN {X 0,Y 429.306,Z 470.987,A -85,B 0,C 180,E1 20365.522,E2 20365.522} C_VEL
LIN {X 0,Y 427.168,Z 466.705,A -85,B 0,C 180,E1 20364.622,E2 20364.622} C_VEL
LIN {X 0,Y 425.51,Z 463.505,A -85,B 0,C 180,E1 20363.928,E2 20363.928} C_VEL
LIN {X 0,Y 425.323,Z 462.508,A -85,B 0,C 180,E1 20363.702,E2 20363.702} C_VEL
LIN {X 0,Y 425.293,Z 462.509,A -85,B 0,C 180,E1 20359.931,E2 20359.931} C_VEL
LIN {X 0,Y 425.318,Z 462.508,A -85,B 0,C 180,E1 20356.105,E2 20356.105} C_VEL
LIN {X 0,Y 425.271,Z 462.514,A -85,B 0,C 180,E1 20352.216,E2 20352.216} C_VEL
LIN {X 0,Y 425.305,Z 462.51,A -85,B 0,C 180,E1 20348.381,E2 20348.381} C_VEL
LIN {X 0,Y 425.306,Z 462.508,A -85,B 0,C 180,E1 20344.72,E2 20344.72} C_VEL
LIN {X 0,Y 425.308,Z 462.504,A -85,B 0,C 180,E1 20340.808,E2 20340.808} C_VEL
LIN {X 0,Y 425.31,Z 462.507,A -85,B 0,C 180,E1 20337.035,E2 20337.035} C_VEL
LIN {X 0,Y 425.325,Z 462.491,A -85,B 0,C 180,E1 20332.978,E2 20332.978} C_VEL
LIN {X 0,Y 425.301,Z 462.507,A -85,B 0,C 180,E1 20329.159,E2 20329.159} C_VEL
LIN {X 0,Y 425.281,Z 462.506,A -85,B 0,C 180,E1 20325.291,E2 20325.291} C_VEL
LIN {X 0,Y 425.315,Z 462.491,A -85,B 0,C 180,E1 20321.496,E2 20321.496} C_VEL
LIN {X 0,Y 425.277,Z 462.496,A -85,B 0,C 180,E1 20317.758,E2 20317.758} C_VEL
LIN {X 0,Y 425.318,Z 462.503,A -85,B 0,C 180,E1 20314.071,E2 20314.071} C_VEL
LIN {X 0,Y 425.288,Z 462.513,A -85,B 0,C 180,E1 20310.415,E2 20310.415} C_VEL
LIN {X 0,Y 425.317,Z 462.507,A -85,B 0,C 180,E1 20306.568,E2 20306.568} C_VEL
LIN {X 0,Y 425.284,Z 462.508,A -85,B 0,C 180,E1 20302.827,E2 20302.827} C_VEL
LIN {X 0,Y 425.292,Z 462.501,A -85,B 0,C 180,E1 20298.79,E2 20298.79} C_VEL
LIN {X 0,Y 425.345,Z 462.677,A -85,B 0,C 180,E1 20295.343,E2 20295.343} C_VEL
LIN {X 0,Y 426.787,Z 466.254,A -85,B 0,C 180,E1 20294.777,E2 20294.777} C_VEL
LIN {X 0,Y 434.019,Z 481.763,A -85,B 0,C 180,E1 20292.274,E2 20292.274} C_VEL
LIN {X 0,Y 441.211,Z 499.039,A -85,B 0,C 180,E1 20289.804,E2 20289.804} C_VEL
LIN {X 0,Y 442.666,Z 501.873,A -85,B 0,C 180,E1 20289.524,E2 20289.524} C_VEL
LIN {X 0,Y 450.156,Z 515.646,A -85,B 0,C 180,E1 20288.458,E2 20288.458} C_VEL
LIN {X 0,Y 452.193,Z 528.44,A -85,B 0,C 180,E1 20287.997,E2 20287.997} C_VEL
LIN {X 0,Y 446.417,Z 760.76,A -85,B 0,C 180,E1 20283.973,E2 20283.973} C_VEL
LIN {X 0,Y 446.206,Z 766.063,A -85,B 0,C 180,E1 20283.851,E2 20283.851} C_VEL
LIN {X 0,Y 444.911,Z 773.664,A -85,B 0,C 180,E1 20283.727,E2 20283.727} C_VEL
LIN {X 0,Y 438.772,Z 792.723,A -85,B 0,C 180,E1 20283.501,E2 20283.501} C_VEL
LIN {X 0,Y 437.32,Z 800.081,A -85,B 0,C 180,E1 20283.255,E2 20283.255} C_VEL
LIN {X 0,Y 435.517,Z 819.392,A -85,B 0,C 180,E1 20282.26,E2 20282.26} C_VEL
LIN {X 0,Y 433.37,Z 838.054,A -85,B 0,C 180,E1 20281.04,E2 20281.04} C_VEL
LIN {X 0,Y 431.031,Z 855.862,A -85,B 0,C 180,E1 20279.609,E2 20279.609} C_VEL
LIN {X 0,Y 428.609,Z 872.823,A -85,B 0,C 180,E1 20277.962,E2 20277.962} C_VEL
LIN {X 0,Y 426.09,Z 889.405,A -85,B 0,C 180,E1 20276.027,E2 20276.027} C_VEL
LIN {X 0,Y 423.75,Z 904.351,A -85,B 0,C 180,E1 20273.943,E2 20273.943} C_VEL
LIN {X 0,Y 421.677,Z 917.815,A -85,B 0,C 180,E1 20271.709,E2 20271.709} C_VEL
LIN {X 0,Y 419.907,Z 929.861,A -85,B 0,C 180,E1 20269.327,E2 20269.327} C_VEL
LIN {X 0,Y 418.408,Z 940.985,A -85,B 0,C 180,E1 20266.663,E2 20266.663} C_VEL
LIN {X 0,Y 417.311,Z 950.441,A -85,B 0,C 180,E1 20263.862,E2 20263.862} C_VEL
LIN {X 0,Y 416.612,Z 957.869,A -85,B 0,C 180,E1 20261.069,E2 20261.069} C_VEL
LIN {X 0,Y 416.23,Z 963.48,A -85,B 0,C 180,E1 20258.286,E2 20258.286} C_VEL
LIN {X 0,Y 416.041,Z 967.417,A -85,B 0,C 180,E1 20255.516,E2 20255.516} C_VEL
LIN {X 0,Y 415.984,Z 969.78,A -85,B 0,C 180,E1 20252.755,E2 20252.755} C_VEL
LIN {X 0,Y 415.98,Z 970.607,A -85,B 0,C 180,E1 20249.999,E2 20249.999} C_VEL
LIN {X 0,Y 415.98,Z 969.823,A -85,B 0,C 180,E1 20247.244,E2 20247.244} C_VEL
LIN {X 0,Y 416.037,Z 967.518,A -85,B 0,C 180,E1 20244.483,E2 20244.483} C_VEL
LIN {X 0,Y 416.225,Z 963.636,A -85,B 0,C 180,E1 20241.712,E2 20241.712} C_VEL
LIN {X 0,Y 416.597,Z 958.082,A -85,B 0,C 180,E1 20238.929,E2 20238.929} C_VEL
LIN {X 0,Y 417.285,Z 950.714,A -85,B 0,C 180,E1 20236.136,E2 20236.136} C_VEL
LIN {X 0,Y 418.365,Z 941.312,A -85,B 0,C 180,E1 20233.333,E2 20233.333} C_VEL
LIN {X 0,Y 419.849,Z 930.244,A -85,B 0,C 180,E1 20230.668,E2 20230.668} C_VEL
LIN {X 0,Y 421.604,Z 918.276,A -85,B 0,C 180,E1 20228.286,E2 20228.286} C_VEL
LIN {X 0,Y 423.669,Z 904.905,A -85,B 0,C 180,E1 20226.05,E2 20226.05} C_VEL
LIN {X 0,Y 425.994,Z 890.064,A -85,B 0,C 180,E1 20223.965,E2 20223.965} C_VEL
LIN {X 0,Y 428.404,Z 874.259,A -85,B 0,C 180,E1 20222.098,E2 20222.098} C_VEL
LIN {X 0,Y 430.82,Z 857.602,A -85,B 0,C 180,E1 20220.45,E2 20220.45} C_VEL
LIN {X 0,Y 433.248,Z 839.219,A -85,B 0,C 180,E1 20218.948,E2 20218.948} C_VEL
LIN {X 0,Y 435.378,Z 820.703,A -85,B 0,C 180,E1 20217.727,E2 20217.727} C_VEL
LIN {X 0,Y 437.218,Z 801.331,A -85,B 0,C 180,E1 20216.711,E2 20216.711} C_VEL
LIN {X 0,Y 438.755,Z 781.147,A -85,B 0,C 180,E1 20215.912,E2 20215.912} C_VEL
LIN {X 0,Y 439.86,Z 760.027,A -85,B 0,C 180,E1 20215.329,E2 20215.329} C_VEL
LIN {X 0,Y 445.549,Z 539.095,A -85,B 0,C 180,E1 20211.447,E2 20211.447} C_VEL
LIN {X 0,Y 439.485,Z 516.498,A -85,B 0,C 180,E1 20210.339,E2 20210.339} C_VEL
LIN {X 0,Y 431.639,Z 502.482,A -85,B 0,C 180,E1 20209.14,E2 20209.14} C_VEL
LIN {X 0,Y 426.265,Z 486.588,A -85,B 0,C 180,E1 20206.214,E2 20206.214} C_VEL
LIN {X 0,Y 421.207,Z 473.389,A -85,B 0,C 180,E1 20203.504,E2 20203.504} C_VEL
LIN {X 0,Y 418.283,Z 466.335,A -85,B 0,C 180,E1 20201.976,E2 20201.976} C_VEL
LIN {X 0,Y 417.376,Z 463.49,A -85,B 0,C 180,E1 20201.338,E2 20201.338} C_VEL
LIN {X 0,Y 417.384,Z 463.514,A -85,B 0,C 180,E1 20200.267,E2 20200.267} C_VEL
LIN {X 0,Y 425.332,Z 484.035,A -85,B 0,C 180,E1 20196.662,E2 20196.662} C_VEL
LIN {X 0,Y 432.152,Z 503.013,A -85,B 0,C 180,E1 20193.571,E2 20193.571} C_VEL
LIN {X 0,Y 435.43,Z 512.991,A -85,B 0,C 180,E1 20192.035,E2 20192.035} C_VEL
LIN {X 0,Y 432.662,Z 546.841,A -85,B 0,C 180,E1 20188.278,E2 20188.278} C_VEL
LIN {X 0,Y 429.962,Z 582.682,A -85,B 0,C 180,E1 20184.379,E2 20184.379} C_VEL
LIN {X 0,Y 427.524,Z 619.333,A -85,B 0,C 180,E1 20180.465,E2 20180.465} C_VEL
LIN {X 0,Y 427.535,Z 621.424,A -85,B 0,C 180,E1 20180.29,E2 20180.29} C_VEL
LIN {X 0,Y 428.169,Z 627.567,A -85,B 0,C 180,E1 20180.1,E2 20180.1} C_VEL
LIN {X 0,Y 423.984,Z 763.049,A -85,B 0,C 180,E1 20176.986,E2 20176.986} C_VEL
LIN {X 0,Y 423.598,Z 779.44,A -85,B 0,C 180,E1 20176.38,E2 20176.38} C_VEL
LIN {X 0,Y 423.01,Z 795.015,A -85,B 0,C 180,E1 20175.562,E2 20175.562} C_VEL
LIN {X 0,Y 422.231,Z 810.504,A -85,B 0,C 180,E1 20174.468,E2 20174.468} C_VEL
LIN {X 0,Y 421.361,Z 824.885,A -85,B 0,C 180,E1 20173.168,E2 20173.168} C_VEL
LIN {X 0,Y 420.411,Z 838.604,A -85,B 0,C 180,E1 20171.594,E2 20171.594} C_VEL
LIN {X 0,Y 419.617,Z 849.693,A -85,B 0,C 180,E1 20170.017,E2 20170.017} C_VEL
LIN {X 0,Y 418.838,Z 860.513,A -85,B 0,C 180,E1 20168.097,E2 20168.097} C_VEL
LIN {X 0,Y 418.26,Z 869.1,A -85,B 0,C 180,E1 20166.176,E2 20166.176} C_VEL
LIN {X 0,Y 417.811,Z 876.659,A -85,B 0,C 180,E1 20163.98,E2 20163.98} C_VEL
LIN {X 0,Y 417.555,Z 881.846,A -85,B 0,C 180,E1 20161.921,E2 20161.921} C_VEL
LIN {X 0,Y 417.452,Z 885.781,A -85,B 0,C 180,E1 20159.589,E2 20159.589} C_VEL
LIN {X 0,Y 417.474,Z 887.67,A -85,B 0,C 180,E1 20157.392,E2 20157.392} C_VEL
LIN {X 0,Y 417.644,Z 887.859,A -85,B 0,C 180,E1 20155.056,E2 20155.056} C_VEL
LIN {X 0,Y 417.943,Z 886.225,A -85,B 0,C 180,E1 20152.854,E2 20152.854} C_VEL
LIN {X 0,Y 418.429,Z 882.905,A -85,B 0,C 180,E1 20150.649,E2 20150.649} C_VEL
LIN {X 0,Y 419.125,Z 877.604,A -85,B 0,C 180,E1 20148.441,E2 20148.441} C_VEL
LIN {X 0,Y 420.004,Z 870.754,A -85,B 0,C 180,E1 20146.369,E2 20146.369} C_VEL
LIN {X 0,Y 421.044,Z 862.36,A -85,B 0,C 180,E1 20144.435,E2 20144.435} C_VEL
LIN {X 0,Y 422.118,Z 853.254,A -85,B 0,C 180,E1 20142.778,E2 20142.778} C_VEL
LIN {X 0,Y 423.422,Z 841.409,A -85,B 0,C 180,E1 20141.053,E2 20141.053} C_VEL
LIN {X 0,Y 424.607,Z 828.745,A -85,B 0,C 180,E1 20139.604,E2 20139.604} C_VEL
LIN {X 0,Y 425.639,Z 815.523,A -85,B 0,C 180,E1 20138.401,E2 20138.401} C_VEL
LIN {X 0,Y 426.543,Z 800.12,A -85,B 0,C 180,E1 20137.319,E2 20137.319} C_VEL
LIN {X 0,Y 427.102,Z 784.491,A -85,B 0,C 180,E1 20136.526,E2 20136.526} C_VEL
LIN {X 0,Y 428.155,Z 754.036,A -85,B 0,C 180,E1 20135.452,E2 20135.452} C_VEL
LIN {X 0,Y 437.255,Z 654.081,A -85,B 0,C 180,E1 20132.157,E2 20132.157} C_VEL
LIN {X 0,Y 444.007,Z 640.226,A -85,B 0,C 180,E1 20130.969,E2 20130.969} C_VEL
LIN {X 0,Y 450.864,Z 617.373,A -85,B 0,C 180,E1 20127.693,E2 20127.693} C_VEL
LIN {X 0,Y 458.181,Z 599.901,A -85,B 0,C 180,E1 20124.976,E2 20124.976} C_VEL
LIN {X 0,Y 466.543,Z 585.323,A -85,B 0,C 180,E1 20122.509,E2 20122.509} C_VEL
LIN {X 0,Y 468.146,Z 583.056,A -85,B 0,C 180,E1 20122.06,E2 20122.06} C_VEL
LIN {X 0,Y 459.831,Z 595.266,A -85,B 0,C 180,E1 20120.332,E2 20120.332} C_VEL
LIN {X 0,Y 453.968,Z 607.33,A -85,B 0,C 180,E1 20118.587,E2 20118.587} C_VEL
LIN {X 0,Y 450.282,Z 619.866,A -85,B 0,C 180,E1 20116.748,E2 20116.748} C_VEL
LIN {X 0,Y 449.093,Z 632.313,A -85,B 0,C 180,E1 20114.893,E2 20114.893} C_VEL
LIN {X 0,Y 450.236,Z 644.513,A -85,B 0,C 180,E1 20113.062,E2 20113.062} C_VEL
LIN {X 0,Y 453.679,Z 656.372,A -85,B 0,C 180,E1 20111.277,E2 20111.277} C_VEL
LIN {X 0,Y 459.29,Z 667.633,A -85,B 0,C 180,E1 20109.588,E2 20109.588} C_VEL
LIN {X 0,Y 466.903,Z 678.307,A -85,B 0,C 180,E1 20107.996,E2 20107.996} C_VEL
LIN {X 0,Y 470.521,Z 682.541,A -85,B 0,C 180,E1 20107.376,E2 20107.376} C_VEL
LIN {X 0,Y 459.111,Z 701.322,A -85,B 0,C 180,E1 20106.706,E2 20106.706} C_VEL
LIN {X 0,Y 450.476,Z 718.35,A -85,B 0,C 180,E1 20105.95,E2 20105.95} C_VEL
LIN {X 0,Y 444.551,Z 732.662,A -85,B 0,C 180,E1 20105.243,E2 20105.243} C_VEL
LIN {X 0,Y 441.422,Z 752.334,A -85,B 0,C 180,E1 20105.146,E2 20105.146} C_VEL
LIN {X 0,Y 439.261,Z 773.721,A -85,B 0,C 180,E1 20104.926,E2 20104.926} C_VEL
LIN {X 0,Y 438.236,Z 804.045,A -85,B 0,C 180,E1 20104.358,E2 20104.358} C_VEL
LIN {X 0,Y 436.874,Z 824.815,A -85,B 0,C 180,E1 20103.746,E2 20103.746} C_VEL
LIN {X 0,Y 435.117,Z 844.679,A -85,B 0,C 180,E1 20102.92,E2 20102.92} C_VEL
LIN {X 0,Y 433.164,Z 863.187,A -85,B 0,C 180,E1 20101.911,E2 20101.911} C_VEL
LIN {X 0,Y 430.898,Z 882.263,A -85,B 0,C 180,E1 20100.612,E2 20100.612} C_VEL
LIN {X 0,Y 428.391,Z 901.016,A -85,B 0,C 180,E1 20099.044,E2 20099.044} C_VEL
LIN {X 0,Y 426.038,Z 918.103,A -85,B 0,C 180,E1 20097.311,E2 20097.311} C_VEL
LIN {X 0,Y 423.809,Z 933.743,A -85,B 0,C 180,E1 20095.429,E2 20095.429} C_VEL
LIN {X 0,Y 421.759,Z 948.47,A -85,B 0,C 180,E1 20093.323,E2 20093.323} C_VEL
LIN {X 0,Y 419.969,Z 961.857,A -85,B 0,C 180,E1 20091.05,E2 20091.05} C_VEL
LIN {X 0,Y 418.527,Z 973.685,A -85,B 0,C 180,E1 20088.671,E2 20088.671} C_VEL
LIN {X 0,Y 417.425,Z 984.778,A -85,B 0,C 180,E1 20085.99,E2 20085.99} C_VEL
LIN {X 0,Y 416.703,Z 993.797,A -85,B 0,C 180,E1 20083.318,E2 20083.318} C_VEL
LIN {X 0,Y 416.303,Z 1000.989,A -85,B 0,C 180,E1 20080.658,E2 20080.658} C_VEL
LIN {X 0,Y 416.145,Z 1006.703,A -85,B 0,C 180,E1 20077.872,E2 20077.872} C_VEL
LIN {X 0,Y 416.1,Z 1010.429,A -85,B 0,C 180,E1 20075.24,E2 20075.24} C_VEL
LIN {X 0,Y 416.135,Z 1012.742,A -85,B 0,C 180,E1 20072.479,E2 20072.479} C_VEL
LIN {X 0,Y 416.158,Z 1013.45,A -85,B 0,C 180,E1 20069.863,E2 20069.863} C_VEL
LIN {X 0,Y 416.128,Z 1012.601,A -85,B 0,C 180,E1 20067.246,E2 20067.246} C_VEL
LIN {X 0,Y 416.096,Z 1010.265,A -85,B 0,C 180,E1 20064.623,E2 20064.623} C_VEL
LIN {X 0,Y 416.129,Z 1006.445,A -85,B 0,C 180,E1 20061.99,E2 20061.99} C_VEL
LIN {X 0,Y 416.303,Z 1000.683,A -85,B 0,C 180,E1 20059.203,E2 20059.203} C_VEL
LIN {X 0,Y 416.73,Z 992.973,A -85,B 0,C 180,E1 20056.401,E2 20056.401} C_VEL
LIN {X 0,Y 417.49,Z 983.73,A -85,B 0,C 180,E1 20053.728,E2 20053.728} C_VEL
LIN {X 0,Y 418.575,Z 973.041,A -85,B 0,C 180,E1 20051.188,E2 20051.188} C_VEL
LIN {X 0,Y 420.13,Z 960.185,A -85,B 0,C 180,E1 20048.647,E2 20048.647} C_VEL
LIN {X 0,Y 421.961,Z 946.589,A -85,B 0,C 180,E1 20046.394,E2 20046.394} C_VEL
LIN {X 0,Y 424.06,Z 931.559,A -85,B 0,C 180,E1 20044.289,E2 20044.289} C_VEL
LIN {X 0,Y 426.45,Z 914.97,A -85,B 0,C 180,E1 20042.34,E2 20042.34} C_VEL
LIN {X 0,Y 428.865,Z 897.297,A -85,B 0,C 180,E1 20040.61,E2 20040.61} C_VEL
LIN {X 0,Y 431.311,Z 878.432,A -85,B 0,C 180,E1 20039.097,E2 20039.097} C_VEL
LIN {X 0,Y 433.486,Z 859.748,A -85,B 0,C 180,E1 20037.883,E2 20037.883} C_VEL
LIN {X 0,Y 435.463,Z 840.198,A -85,B 0,C 180,E1 20036.876,E2 20036.876} C_VEL
LIN {X 0,Y 437.159,Z 819.613,A -85,B 0,C 180,E1 20036.078,E2 20036.078} C_VEL
LIN {X 0,Y 438.407,Z 798.926,A -85,B 0,C 180,E1 20035.524,E2 20035.524} C_VEL
LIN {X 0,Y 439.515,Z 768.342,A -85,B 0,C 180,E1 20034.997,E2 20034.997} C_VEL
LIN {X 0,Y 441.354,Z 751.007,A -85,B 0,C 180,E1 20034.792,E2 20034.792} C_VEL
LIN {X 0,Y 448.195,Z 734.76,A -85,B 0,C 180,E1 20033.919,E2 20033.919} C_VEL
LIN {X 0,Y 456.206,Z 716.894,A -85,B 0,C 180,E1 20033.015,E2 20033.015} C_VEL
LIN {X 0,Y 465.87,Z 699.333,A -85,B 0,C 180,E1 20032.29,E2 20032.29} C_VEL
LIN {X 0,Y 473.925,Z 686.251,A -85,B 0,C 180,E1 20031.83,E2 20031.83} C_VEL
LIN {X 0,Y 465.342,Z 675.379,A -85,B 0,C 180,E1 20030.283,E2 20030.283} C_VEL
LIN {X 0,Y 457.67,Z 662.033,A -85,B 0,C 180,E1 20028.533,E2 20028.533} C_VEL
